KUKA KRL program: vw_sz_usr_s.src, vw_sz_usr_s.dat

--- vw_sz_usr_s.src ---
&ACCESS RV
&REL 203
&PARAM DISKPATH = VW_User/Applikation/S_Zange
&PARAM TPVW_VERSION = 8.3.0
DEF vw_sz_usr_s( )
;
;*-----------------------------------------------------*
;*Technologiepaket S_Zangen                            *
;*                                                     *
;*Konzernstandard                                      *
;*Bearbeiter: W. Lehmeier I/PG-C61                     *
;*                                                     *
;* Erstellt am:                                        *
;* 2015.02.19 LE                                       *
;* 2017.01.26 MBA Anpassung Teachfunktion KE           *
;* 2017.02.03 MBA Mit_BM1 bei BM2 korrigiert           *
;*            Zangenfkt. bei BM2 korrigiert            *
;* 2017.09.26 LZ "F_SZ_POT_Fra=838" bei POT gegen      *
;*            "Prog_Nr_SZ#>98" getauscht               *
;*                                                     *
;*------------------------------------------------------
;
END
;
;FOLD INIT S_Zangen
GLOBAL DEF SZ_INIT( )
INT i
;
;FOLD Version Techpaket
Tech_S_Zangen.Name[]="KS24.01.008_170926"
;ENDFOLD
;
;FOLD Vorbesetzung Meldungsausgabe
FOR i = 1 TO 100
  n_SZS_Handle[i]=-1
  n_SZR_Handle[i]=-1
ENDFOR
;ENDFOLD
;
;FOLD TimerInit
FOR i = 1 TO 3
  LBitTimeCnt[i] = $Rob_Timer
ENDFOR
;ENDFOLD
;
; Zaehle Flags fuer q-Tool
;SZ1
IF $Flag[F_QT_SZ1_VW] THEN
  Q_T_SZ1_VW=Q_T_SZ1_VW+1
ENDIF
IF $Flag[F_QT_SZ1_Fe] THEN
  Q_T_SZ1_Fe=Q_T_SZ1_Fe+1
ENDIF
IF $Flag[F_QT_SZ1_kD] THEN
  Q_T_SZ1_kD=Q_T_SZ1_kD+1
ELSE
  Q_T_SZ1_kD=0
ENDIF
;
;SZ2
IF $Flag[F_QT_SZ2_VW] THEN
  Q_T_SZ2_VW=Q_T_SZ2_VW+1
ENDIF
IF $Flag[F_QT_SZ2_Fe] THEN
  Q_T_SZ2_Fe=Q_T_SZ2_Fe+1
ENDIF
IF $Flag[F_QT_SZ2_kD] THEN
  Q_T_SZ2_kD=Q_T_SZ2_kD+1
ELSE
  Q_T_SZ2_kD=0
ENDIF
;SZ3
;
IF $Flag[F_QT_SZ3_VW] THEN
  Q_T_SZ3_VW=Q_T_SZ3_VW+1
ENDIF
IF $Flag[F_QT_SZ3_Fe] THEN
  Q_T_SZ3_Fe=Q_T_SZ3_Fe+1
ENDIF
IF $Flag[F_QT_SZ3_kD] THEN
  Q_T_SZ3_kD=Q_T_SZ3_kD+1
ELSE
  Q_T_SZ3_kD=0
ENDIF
;
; Zaehlergrenze damit kein ueberlauf entsteht
IF Q_T_SZ1_VW>1000000 THEN
  Q_T_SZ1_VW=0
ENDIF
IF Q_T_SZ1_Fe>1000000 THEN
  Q_T_SZ1_Fe=0
ENDIF
IF Q_T_SZ1_kD>1000000 THEN
  Q_T_SZ1_kD=0
ENDIF
IF Q_T_SZ2_VW>1000000 THEN
  Q_T_SZ2_VW=0
ENDIF
IF Q_T_SZ2_Fe>1000000 THEN
  Q_T_SZ2_Fe=0
ENDIF
IF Q_T_SZ2_kD>1000000 THEN
  Q_T_SZ2_kD=0
ENDIF
IF Q_T_SZ3_VW>1000000 THEN
  Q_T_SZ3_VW=0
ENDIF
IF Q_T_SZ3_Fe>1000000 THEN
  Q_T_SZ3_Fe=0
ENDIF
IF Q_T_SZ3_kD>1000000 THEN
  Q_T_SZ3_kD=0
ENDIF
;
$FLAG[F_QT_SZ1_VW]=FALSE
$FLAG[F_QT_SZ1_Fe]=FALSE
$FLAG[F_QT_SZ1_kD]=FALSE
$FLAG[F_QT_SZ2_VW]=FALSE
$FLAG[F_QT_SZ2_Fe]=FALSE
$FLAG[F_QT_SZ2_kD]=FALSE
$FLAG[F_QT_SZ3_VW]=FALSE
$FLAG[F_QT_SZ3_Fe]=FALSE
$FLAG[F_QT_SZ3_kD]=FALSE
;
;FOLD Vorbesetzung SZ1-3
IF $PRO_STATE1==#P_FREE THEN
  IF ($softplcint[2]>0) AND (NOT Docking OR DKSZ_stat_SZ) THEN
    I_SZ2_bereit=865
    O_SZ2_FRG=875
    I_SZ2_aktiv=875
    O_SZ2_SPos_g=876
    I_SZ2_IPos_g=876
    I_SZ2_F_Ziel=933
    ;Docking Downgrade
    bhf3_belegt=4081
    bhf4_belegt=4081
  ENDIF
  IF ($softplcint[3]>0) AND (NOT Docking OR DKSZ_stat_SZ) THEN
    I_SZ3_bereit=1025
    O_SZ3_FRG=1035
    I_SZ3_aktiv=1035
    O_SZ3_SPos_g=1036
    I_SZ3_IPos_g=1036
    I_SZ3_F_Ziel=1093
    ;Docking Downgrade
    bhf3_belegt=559
    bhf4_belegt=4081
  ENDIF
  IF Docking AND NOT DOCK_SP AND NOT DKSZ_stat_SZ THEN
    I_SZ2_bereit=4081
    O_SZ2_FRG=3658
    I_SZ2_aktiv=4082
    O_SZ2_SPos_g=3658
    I_SZ2_IPos_g=4081
    I_SZ2_F_Ziel=4082
    I_SZ3_bereit=4081
    O_SZ3_FRG=3658
    I_SZ3_aktiv=4082
    O_SZ3_SPos_g=3658
    I_SZ3_IPos_g=4081
    I_SZ3_F_Ziel=4082
    ;Docking Downgrade
    IF (AX_SIM_ON=='B000111000000') OR (AX_SIM_ON=='B001110000000') THEN
      bhf3_belegt=559
    ENDIF
    IF (AX_SIM_ON=='B001111000000') OR (AX_SIM_ON=='B011110000000') THEN
      bhf4_belegt=560
    ENDIF
  ENDIF
ENDIF
;ENDFOLD (Vorbesetzung SZ1-3)
;
;Ausgleichsfunktion initialisieren
R1AusgleichFunktion=0
GunBal_Halt=FALSE
;
;Hilfsflag fuer SZ-AH-Kompensation ausschalten
$FLAG[F_SZ_AH_KOMP]=FALSE
;Hilfsflag fuer SZ_Schliessen ausschalten
$FLAG[F_SZ1_Schliess]=FALSE
$FLAG[F_SZ2_Schliess]=FALSE
$FLAG[F_SZ3_Schliess]=FALSE
;
;Initiallisierung Kappenstandzeit Z1-3
FOR i = 1 TO 10
  IF (ReserveReal[i]==0.0) THEN
    ReserveReal[i]=28.0
  ENDIF
ENDFOR
;
END
;ENDFOLD
;
;-----------------------------------------------------------
;FOLD SAW S_Zangen
GLOBAL DEF SZ_SAW( )
INT i
;
;FOLD S_Zangen 1-3
IF ($softplcint[1]>0) AND NOT ($OUT[O_SZ1_Re_aus] OR $OUT[O_SZ1_MnFrae] OR $OUT[O_Kb1_MnFrae] OR $FLAG[F_SZ1_FRG_FR]) THEN
  $OUT[O_SZ1_S_TPos]=FALSE
  $OUT[O_SZ1_ref]=FALSE
  $OUT[O_SZ1_FRG]=FALSE
  $OUT[O_SZ1_auf]=FALSE
  $OUT[O_SZ1_zu]=FALSE
  $OUT[O_SZ1_t_auf]=FALSE
  $OUT[O_SZ1_t_zu]=FALSE
  IF Mit_Komb_ST1 THEN
    $OUT[O_Kb1_t_auf]=FALSE
    $OUT[O_Kb1_t_zu]=FALSE
  ENDIF
ENDIF
IF ($softplcint[2]>0) AND NOT ($OUT[O_SZ2_Re_aus] OR $OUT[O_SZ2_MnFrae] OR $OUT[O_Kb2_MnFrae] OR $FLAG[F_SZ2_FRG_FR]) THEN
  $OUT[O_SZ2_S_TPos]=FALSE
  $OUT[O_SZ2_ref]=FALSE
  $OUT[O_SZ2_FRG]=FALSE
  $OUT[O_SZ2_auf]=FALSE
  $OUT[O_SZ2_zu]=FALSE
  $OUT[O_SZ2_t_auf]=FALSE
  $OUT[O_SZ2_t_zu]=FALSE
  IF Mit_Komb_ST2 THEN
    $OUT[O_Kb2_t_auf]=FALSE
    $OUT[O_Kb2_t_zu]=FALSE
  ENDIF
ENDIF
IF ($softplcint[3]>0) AND NOT ($OUT[O_SZ3_Re_aus] OR $OUT[O_SZ3_MnFrae] OR $OUT[O_Kb3_MnFrae] OR $FLAG[F_SZ3_FRG_FR]) THEN
  $OUT[O_SZ3_S_TPos]=FALSE
  $OUT[O_SZ3_ref]=FALSE
  $OUT[O_SZ3_FRG]=FALSE
  $OUT[O_SZ3_auf]=FALSE
  $OUT[O_SZ3_zu]=FALSE
  $OUT[O_SZ3_t_auf]=FALSE
  $OUT[O_SZ3_t_zu]=FALSE
  IF Mit_Komb_ST3 THEN
    $OUT[O_Kb3_t_auf]=FALSE
    $OUT[O_Kb3_t_zu]=FALSE
  ENDIF
ENDIF
HAND_FKT1=FALSE
HAND_FKT2=FALSE
;
;SZ Ausgleich durch Roboter
IF R1AusgleichFunktion>0 THEN
  R1AusgleichFunktion=0
  S_Zangen_Msg(20,#NotifyMsg)
ENDIF
GunBal_Halt=FALSE
;
;Hilfsflag fuer SZ-AH-Kompensation ausschalten
$FLAG[F_SZ_AH_KOMP]=FALSE
;Hilfsflag fuer SZ_Schliessen ausschalten
$FLAG[F_SZ1_Schliess]=FALSE
$FLAG[F_SZ2_Schliess]=FALSE
$FLAG[F_SZ3_Schliess]=FALSE
;ENDFOLD
;
END
;ENDFOLD
;
;-----------------------------------------------------------
;FOLD RESET S_Zangen
GLOBAL DEF SZ_RESET( )
INT i
;
;FOLD S_Zangen 1-3
IF (($mode_op==#T1) OR ($mode_op==#T2)) THEN
  $softplcint[20]=0
  IF ($softplcint[1]>0) THEN
    $FLAG[F_SZ_AH_KOMP]=FALSE
    $OUT[O_SZ1_FRG]=FALSE
    $OUT[O_SZ1_S_TPos]=FALSE
    $OUT[O_SZ1_ref]=FALSE
    $OUT[O_SZ1_auf]=FALSE
    $OUT[O_SZ1_zu]=FALSE
    $OUT[O_SZ1_t_auf]=FALSE
    $OUT[O_SZ1_t_zu]=FALSE
    $OUT[O_SZ1_MvFrae]=FALSE
    $OUT[O_SZ1_MnFrae]=FALSE
    IF Mit_Komb_ST1 THEN
      $OUT[O_Kb1_t_auf]=FALSE
      $OUT[O_Kb1_t_zu]=FALSE
    ENDIF
  ENDIF
;
  IF ($softplcint[2]>0) THEN
    $OUT[O_SZ2_FRG]=FALSE
    $OUT[O_SZ2_S_TPos]=FALSE
    $OUT[O_SZ2_ref]=FALSE
    $OUT[O_SZ2_auf]=FALSE
    $OUT[O_SZ2_zu]=FALSE
    $OUT[O_SZ2_t_auf]=FALSE
    $OUT[O_SZ2_t_zu]=FALSE
    $OUT[O_SZ2_MvFrae]=FALSE
    $OUT[O_SZ2_MnFrae]=FALSE
    IF Mit_Komb_ST2 THEN
      $OUT[O_Kb2_t_auf]=FALSE
      $OUT[O_Kb2_t_zu]=FALSE
    ENDIF
  ENDIF
;
  IF ($softplcint[3]>0) THEN
    $OUT[O_SZ3_FRG]=FALSE
    $OUT[O_SZ3_S_TPos]=FALSE
    $OUT[O_SZ3_ref]=FALSE
    $OUT[O_SZ3_auf]=FALSE
    $OUT[O_SZ3_zu]=FALSE
    $OUT[O_SZ3_t_auf]=FALSE
    $OUT[O_SZ3_t_zu]=FALSE
    $OUT[O_SZ3_MvFrae]=FALSE
    $OUT[O_SZ3_MnFrae]=FALSE
    IF Mit_Komb_ST3 THEN
      $OUT[O_Kb3_t_auf]=FALSE
      $OUT[O_Kb3_t_zu]=FALSE
    ENDIF
  ENDIF
;
  ;SZ Ausgleich durch Roboter
  R1AusgleichFunktion=0
  GunBal_Halt=FALSE
;
  ;Hilfsflag fuer SZ-AH-Kompensation ausschalten
  $FLAG[F_SZ_AH_KOMP]=FALSE
  ;Hilfsflag fuer SZ_Schliessen ausschalten
  $FLAG[F_SZ1_Schliess]=FALSE
  $FLAG[F_SZ2_Schliess]=FALSE
  $FLAG[F_SZ3_Schliess]=FALSE
ENDIF ;(SZ_VORHANDEN)
;ENDFOLD
;
END
;ENDFOLD
;
;-----------------------------------------------------------
;FOLD CANCEL S_Zangen
GLOBAL DEF SZ_CANCEL( )
INT i
;
;FOLD S_Zangen 1-3
IF (($mode_op==#T1) OR ($mode_op==#T2)) THEN
  $softplcint[20]=0
  IF ($softplcint[1]>0) THEN
    $FLAG[F_SZ_AH_KOMP]=FALSE
    $OUT[O_SZ1_FRG]=FALSE
    $OUT[O_SZ1_S_TPos]=FALSE
    $OUT[O_SZ1_ref]=FALSE
    $OUT[O_SZ1_auf]=FALSE
    $OUT[O_SZ1_zu]=FALSE
    $OUT[O_SZ1_t_auf]=FALSE
    $OUT[O_SZ1_t_zu]=FALSE
    $OUT[O_SZ1_MvFrae]=FALSE
    $OUT[O_SZ1_MnFrae]=FALSE
    IF Mit_Komb_ST1 THEN
      $OUT[O_Kb1_t_auf]=FALSE
      $OUT[O_Kb1_t_zu]=FALSE
    ENDIF
  ENDIF
;
  IF ($softplcint[2]>0) THEN
    $OUT[O_SZ2_FRG]=FALSE
    $OUT[O_SZ2_S_TPos]=FALSE
    $OUT[O_SZ2_ref]=FALSE
    $OUT[O_SZ2_auf]=FALSE
    $OUT[O_SZ2_zu]=FALSE
    $OUT[O_SZ2_t_auf]=FALSE
    $OUT[O_SZ2_t_zu]=FALSE
    $OUT[O_SZ2_MvFrae]=FALSE
    $OUT[O_SZ2_MnFrae]=FALSE
    IF Mit_Komb_ST2 THEN
      $OUT[O_Kb2_t_auf]=FALSE
      $OUT[O_Kb2_t_zu]=FALSE
    ENDIF
  ENDIF
;
  IF ($softplcint[3]>0) THEN
    $OUT[O_SZ3_FRG]=FALSE
    $OUT[O_SZ3_S_TPos]=FALSE
    $OUT[O_SZ3_ref]=FALSE
    $OUT[O_SZ3_auf]=FALSE
    $OUT[O_SZ3_zu]=FALSE
    $OUT[O_SZ3_t_auf]=FALSE
    $OUT[O_SZ3_t_zu]=FALSE
    $OUT[O_SZ3_MvFrae]=FALSE
    $OUT[O_SZ3_MnFrae]=FALSE
    IF Mit_Komb_ST3 THEN
      $OUT[O_Kb3_t_auf]=FALSE
      $OUT[O_Kb3_t_zu]=FALSE
    ENDIF
  ENDIF
;
  ;SZ Ausgleich durch Roboter
  R1AusgleichFunktion=0
  GunBal_Halt=FALSE
;
  ;Hilfsflag fuer SZ-AH-Kompensation ausschalten
  $FLAG[F_SZ_AH_KOMP]=FALSE
  ;Hilfsflag fuer SZ_Schliessen ausschalten
  $FLAG[F_SZ1_Schliess]=FALSE
  $FLAG[F_SZ2_Schliess]=FALSE
  $FLAG[F_SZ3_Schliess]=FALSE
ENDIF ;(SZ_VORHANDEN)
;ENDFOLD
;
END
;ENDFOLD
;
;-----------------------------------------------------------
;FOLD LOOP S_Zange 1
GLOBAL DEF SZ1_LOOP( )
;
;SZ 1 Funktionstest ohne Bauteil
IF Mit_Komb_ST1 THEN
  $OUT[O_Kb1_FToBT]=$IN[I_FT_o_BT]
  IF (Prog_Nr_Kb1<99) AND ($FLAG[F_SZ1_FRG_FR] OR $OUT[O_R_Wart] OR $OUT[O_R_WartB]) THEN
    Fzg_Typ_SZ1=0
  ENDIF
ELSE
  $OUT[O_SZ1_FToBT]=$IN[I_FT_o_BT] AND (Prog_Nr_SZ1>98)
  IF (Prog_Nr_SZ1<99) AND ($FLAG[F_SZ1_FRG_FR] OR $OUT[O_R_Wart] OR $OUT[O_R_WartB]) THEN
    Fzg_Typ_SZ1=0
	 SK1_Fzg_Typ=0
  ENDIF
ENDIF
;
;SZ 1 Anwahl Energiesparmodus
$OUT[O_SZ1_E_Mode] = (($Brake_Sig==0) AND $timer_flag[TimerNr_E_Mo] AND e_Mode_Hilf2)
;
;FOLD SZ Betriebsarten
;BA-Hand an SZ 1 setzen
IF $OUT[O_R_Hand] AND (NOT $COULD_START_MOTION OR HAND_FKT2) THEN
  $OUT[O_SZ1_R_Hand]=TRUE
  $OUT[O_SZ1_R_Auto]=FALSE
ENDIF
;
;BA-AUTO an SZ 1 setzen
IF $OUT[O_R_Hand] AND NOT HAND_FKT2 AND ($OUT[O_R_Proz_akt] OR $OUT[O_R_bewegt] OR TAST_AKTIV_1 OR TAST_AKTIV_2 OR TAST_AKTIV_3 OR HAND_FKT1) AND (R1AusgleichFunktion==0) OR $OUT[O_R_Auto] THEN
  $OUT[O_SZ1_R_Hand]=FALSE
  $OUT[O_SZ1_R_Auto]=TRUE
ENDIF
;ENDFOLD
;
;SZ 1 mit EK-Verschleisswert
$OUT[O_SZ1_Mit_EK]=TRUE
;
;SZ 1 ohne Kraft
IF $IN[I_SZ1_oh_Kra] THEN
  $OUT[O_SZ1_oh_Kra]=TRUE
ELSE
  $OUT[O_SZ1_oh_Kra]=FALSE
ENDIF
;
;SZ Kraftvorgabe in Hand
IF NOT Mit_Komb_ST1  THEN
  IF $OUT[O_R_Hand] AND $FLAG[F_o_Prozess] THEN
    SZ1_Kraft_Soll = M_Kraft_Soll
  ELSE
    SZ1_Kraft_Soll = SK1_Kraft_Soll
  ENDIF
ENDIF
;ENDFOLD
;
;Kompensation der EK durch Roboter
IF AH_Komp AND NOT $FLAG[F_SZ1_m_Komp] AND NOT Mit_Komb_ST1 THEN
  $OUT[O_SZ1_m_RKom]=TRUE
ELSE
  $OUT[O_SZ1_m_RKom]=FALSE
ENDIF
;
;Quittierung Stoerung
IF Mit_Komb_ST1 THEN
  $OUT[O_Kb1_Fe_Res]=($IN[I_Kb1_Sammel] AND $IN[I_R_Quit_St]) OR (($IN[I_R_Quit_Wei] OR $FLAG[F_SZ_Fe_Res]) AND $IN[I_Kb1_Sammel])
ELSE
  $OUT[O_SZ1_Fe_Res]=($IN[I_SZ1_Sammel] AND $IN[I_R_Quit_St]) OR (($IN[I_R_Quit_Wei] OR $FLAG[F_SZ_Fe_Res]) AND $IN[I_SZ1_Sammel])
ENDIF
;
;Ausgabe Statusmeldungen an BMS
IF Mit_Komb_ST1 THEN
  ;Vorwahl mit Strom
  $OUT[O_Kb1_m_Stro]=NOT $IN[I_Kb1_o_Schw] AND NOT $FLAG[F_o_Prozess]
  ;Start Protokoll
  $OUT[O_Kb1_Protok]=$IN[I_Kb1_Protok]
  ;Vorwarnung Zange
  $OUT[O_Kb1_W_SZ]=($IN[I_SZ1_W_SZ] OR (Q_T_SZ1_VW>3) OR (Q_T_SZ1_kD>50))
  ;Warnung Schmierung
  $OUT[O_Kb1_W_Schm]=$IN[I_SZ1_W_Schm]
  ;Fraesanfrage
  $OUT[O_Kb1_FrAnf]=$OUT[O_R_Auto] AND $IN[I_Kb1_FrAnf]
  ;Vorwarnung Kappenstandzeit
  $OUT[O_Kb1_V_Stdm]=($IN[I_Kb1_V_Stdm] OR B_SK1_V_Stdm)
  ;Maximale Kappenstandzeit
  $OUT[O_Kb1_M_Stdm]=($IN[I_SZ1_F_Geom] OR $IN[I_Kb1_M_Stdm] OR B_SK1_M_Stdm OR $FLAG[F_SK1_max_SZ1] OR $FLAG[F_SK1_max_SZ2] OR $FLAG[F_SK1_max_SZ3] OR $FLAG[F_SK1_max_SZ4])
  ;Kraftaufbau zu lange
  $OUT[O_Kb1_F_Kraf]=$OUT[O_R_Auto] AND $IN[I_SZ1_F_Kraf]
  ;Punktanwahlfehler
  $OUT[O_Kb1_F_Prog]=$OUT[O_R_Auto] AND $IN[I_SZ1_F_Prog]
  ;Zielposition ungueltig
  $OUT[O_Kb1_F_Ziel]=$OUT[O_R_Auto] AND $IN[I_SZ1_F_Ziel]
  ;Bauteilfehler
  $OUT[O_Kb1_F_Baut]=$OUT[O_R_Auto] AND $IN[I_SZ1_F_Baut]
  ;Zange geht schwer
  $OUT[O_Kb1_F_schw]=$OUT[O_R_Auto] AND $IN[I_SZ1_F_schw]
  ;Fraesen n.i.O.
  $OUT[O_Kb1_F_Frae]=$OUT[O_R_Auto] AND $IN[I_SZ1_F_Frae]
  ;Fehler Kappenverschleiss
  $OUT[O_Kb1_F_KaVe]=$OUT[O_R_Auto] AND ($IN[I_SZ1_F_Kapp] OR $FLAG[F_SZ1_Kapp1] OR $FLAG[F_SZ1_Kapp2] OR $FLAG[F_SZ1_Kapp3] OR $FLAG[F_SZ1_Kapp4])
  ;Fehler Geometrie
  $OUT[O_Kb1_F_Geom]=$OUT[O_R_Auto] AND $IN[I_SZ1_F_Geom]
  ;Schleppfehler
  $OUT[O_Kb1_Schlep]=$OUT[O_R_Auto] AND $IN[I_SZ1_F_Schl]
  ;Fehler Ausgleichssystem
  $OUT[O_Kb1_F_Ausg]=$OUT[O_R_Auto] AND ($IN[I_SZ1_F_Ausg] OR (Q_T_SZ1_Fe>3))
  ;Fehler Steuerung/Regler
  $OUT[O_Kb1_F_Steu]=$OUT[O_R_Auto] AND $COULD_START_MOTION AND $IN[I_SZ1_F_Steu]
  ;Fehler Temperatur Trafo
  $OUT[O_Kb1_FT_Tra]=$OUT[O_R_Auto] AND $IN[I_SZ1_F_Traf]
  ;Fehler Temperatur Motor
  $OUT[O_Kb1_FT_Mot]=$OUT[O_R_Auto] AND $IN[I_SZ1_F_Mot]
  ;Schweissung i.O
  $OUT[O_Kb1_WPS_io]=$OUT[O_R_Auto] AND NOT $FLAG[F_SK1_S_niO]
  ;Schweissung n.i.O
  $OUT[O_Kb1_WP_nio]=$OUT[O_R_Auto] AND $FLAG[F_SK1_S_niO]
  ;Warngrenze verletzt in Folge
  $OUT[O_Kb1_W_Folg]=$OUT[O_R_Auto] AND $IN[I_Kb1_W_Folg]
  ;Phasenueberwachung
  $OUT[O_Kb1_Ph_nio]=$OUT[O_R_Auto] AND $IN[I_Kb1_Ph_nio]
  ;Ueberstrom Primaerseite
  $OUT[O_Kb1_Primae]=$OUT[O_R_Auto] AND $IN[I_Kb1_Primae]
  ;Fehler Stromsensor
  $OUT[O_Kb1_F_Stro]=$OUT[O_R_Auto] AND $IN[I_Kb1_F_Stro]
  ;Fehler Spannungssensor
  $OUT[O_Kb1_F_Span]=$OUT[O_R_Auto] AND $IN[I_Kb1_F_Span]
  ;Überstrom 24 V DC
  $OUT[O_Kb1_24V]=$OUT[O_R_Auto] AND $IN[I_Kb1_24V]
  ;Uebertemperatur Inverter
  $OUT[O_Kb1_Invert]=$OUT[O_R_Auto] AND $IN[I_Kb1_Invert]
  ;Sammelstoerung
  $OUT[O_Kb1_Sammel]=$OUT[O_R_Auto] AND $COULD_START_MOTION AND ($IN[I_Kb1_Sammel] OR $FLAG[F_SZ1_Sammel] OR $FLAG[F_SK1_Sammel] OR SZ_LBitFeh[1]) AND $timer_flag[TimerNr_Ein]
ELSE
  ;Vorwarnung Zange
  $OUT[O_SZ1_W_SZ]=($IN[I_SZ1_W_SZ] OR (Q_T_SZ1_VW>3) OR (Q_T_SZ1_kD>50))
  ;Warnung Schmierung
  $OUT[O_SZ1_W_Schm]=$IN[I_SZ1_W_Schm]
  ;Kraftaufbau zu lange
  $OUT[O_SZ1_F_Kraf]=$OUT[O_R_Auto] AND $IN[I_SZ1_F_Kraf]
  ;Programmfehler/falsche Kraftvorgabe
  $OUT[O_SZ1_F_Prog]=$OUT[O_R_Auto] AND $IN[I_SZ1_F_Prog]
  ;Zielposition ungueltig
  $OUT[O_SZ1_F_Ziel]=$OUT[O_R_Auto] AND $IN[I_SZ1_F_Ziel]
  ;Bauteilfehler
  $OUT[O_SZ1_F_Baut]=$OUT[O_R_Auto] AND $IN[I_SZ1_F_Baut]
  ;Zange geht schwer
  $OUT[O_SZ1_F_schw]=$OUT[O_R_Auto] AND $IN[I_SZ1_F_schw]
  ;Fraesen n.i.O.
  $OUT[O_SZ1_F_Frae]=$OUT[O_R_Auto] AND $IN[I_SZ1_F_Frae]
  ;Fehler Kappenverschleiss/Geometrie
  $OUT[O_SZ1_F_Geom]=$OUT[O_R_Auto] AND ($IN[I_SZ1_F_Kapp] OR $IN[I_SZ1_F_Geom] OR $FLAG[F_SZ1_Kapp1] OR $FLAG[F_SZ1_Kapp2] OR $FLAG[F_SZ1_Kapp3] OR $FLAG[F_SZ1_Kapp4])
  ;Fehler Ausgleichssystem
  $OUT[O_SZ1_F_Ausg]=$OUT[O_R_Auto] AND ($IN[I_SZ1_F_Ausg] OR (Q_T_SZ1_Fe>3))
  ;Fehler Steuerung/Regler
  $OUT[O_SZ1_F_Steu]=$OUT[O_R_Auto] AND $COULD_START_MOTION AND $IN[I_SZ1_F_Steu]
  ;Fehler Temperatur Motor/Trafo
  $OUT[O_SZ1_F_Temp]=$OUT[O_R_Auto] AND ($IN[I_SZ1_F_Traf] OR $IN[I_SZ1_F_Mot])
  ;Sammelstoerung
  $OUT[O_SZ1_Sammel]=$OUT[O_R_Auto] AND $COULD_START_MOTION AND ($IN[I_SZ1_Sammel] OR $FLAG[F_SZ1_Sammel] OR SZ_LBitFeh[1]) AND $timer_flag[TimerNr_Ein]
ENDIF
;
;Ausgabe Zangencode
IF NOT Docking OR (Docking AND NOT Dock_SZ) THEN
  IF Mit_Komb_ST THEN
    Kb1_ZCode=1
  ELSE
    EZ1_ZCode=1
  ENDIF
ENDIF
;
;FOLD SZ-Tastbetrieb ruecksetzen
IF Mit_Komb_ST1 THEN
  Temp_Komb_1=($OUT[O_Kb1_t_zu] OR $OUT[O_Kb1_t_auf])
ENDIF
IF $OUT[O_R_Hand] AND TAST_AKTIV_1 AND NOT $OUT[O_SZ1_t_auf] AND NOT $OUT[O_SZ1_t_zu] AND NOT Temp_Komb_1 THEN
  TAST_AKTIV_1=FALSE
  $OUT[O_SZ1_FRG]=FALSE
  schleppfehler=TRUE
  sf_prog_status=#user_act
  $OUT[O_SZ1_SPos_g]=FALSE
ENDIF
;ENDFOLD
;
;FOLD SZ INIT Zangenfunktion
IF $OUT[O_R_Hand] AND NOT $OUT[O_R_Auto] AND $COULD_START_MOTION AND ((NOT $OUT[O_R_Proz_akt] AND NOT $OUT[O_R_bewegt]) OR (R1AusgleichFunktion>0)) THEN
  IF Mit_Komb_ST1 THEN
    Temp_Komb_1=$OUT[O_Kb1_t_zu]
  ENDIF
  IF ($OUT[O_SZ1_S_TPos] OR $OUT[O_SZ1_ref] OR $OUT[O_SZ1_auf] OR $OUT[O_SZ1_zu] OR Temp_Komb_1 OR $OUT[O_SZ1_t_auf] OR $OUT[O_SZ1_t_zu] OR $OUT[O_SZ1_Teach] OR $OUT[O_SZ1_D_Auf] OR $OUT[O_SZ1_Du_Zu]) THEN
    CheckZangenFunktion()
    Zangenfunktion()
  ENDIF
ELSE
  IF $OUT[O_SZ1_Teach] OR $OUT[O_SZ1_D_Auf] OR $OUT[O_SZ1_Du_Zu] THEN
    $OUT[O_SZ1_Teach]=FALSE
    $OUT[O_SZ1_D_Auf]=FALSE
    $OUT[O_SZ1_Du_Zu]=FALSE
    S_Zangen_Msg(34,#NotifyMsg)
  ENDIF
ENDIF
;ENDFOLD
;
;FOLD Ruecksetzen Zangenfunktion
IF ($OUT[O_R_Hand] AND ($PRO_MODE1==#BSTEP)) OR ($OUT[O_R_Hand] AND NOT $FLAG[F_SZ_AH_KOMP] AND $OUT[O_R_bewegt] AND (R1AusgleichFunktion==0)) OR ($OUT[O_R_Hand] AND NOT $COULD_START_MOTION AND (HAND_FKT1 OR HAND_FKT2)) THEN
  IF NOT ($OUT[O_SZ1_Re_aus] OR $OUT[O_SZ1_MnFrae] OR $OUT[O_Kb1_MnFrae] OR $FLAG[F_SZ1_FRG_FR]) THEN
    $OUT[O_SZ1_S_TPos]=FALSE
    $OUT[O_SZ1_ref]=FALSE
    $OUT[O_SZ1_FRG]=FALSE
    $OUT[O_SZ1_auf]=FALSE
    $OUT[O_SZ1_zu]=FALSE
    $OUT[O_SZ1_t_auf]=FALSE
    $OUT[O_SZ1_t_zu]=FALSE
    IF Mit_Komb_ST1 THEN
      $OUT[O_Kb1_t_auf]=FALSE
      $OUT[O_Kb1_t_zu]=FALSE
    ENDIF
  ENDIF
  HAND_FKT1=FALSE
  HAND_FKT2=FALSE
ENDIF
;ENDFOLD
;
;FOLD EZ Oeffnungsmass beim Schwenken pruefen
;EZ/SP1
IF ($softplcint[1]>0) AND $OUT[O_SZ1_FRG] AND (Varstate("act_P1")==#initialized) THEN
  IF ($softplcint[1]==7) THEN
    $FLAG[F_SZ1_Oeff_iO]=(act_P1.E1>=$COUNT_I[60])
  ENDIF
  IF ($softplcint[1]==8) THEN
    $FLAG[F_SZ1_Oeff_iO]=(act_P1.E2>=$COUNT_I[60])
  ENDIF
ELSE
  $FLAG[F_SZ1_Oeff_iO]=FALSE
ENDIF
;ENDFOLD
;
;FOLD EZ Position nach Messen und Fraesen pruefen
$FLAG[Mit_Anf_Pos]=TRUE
;EZ/SP1
IF ($softplcint[1]>0) AND $FLAG[F_SZ_Anf_Pos] AND $OUT[O_SZ1_FRG] AND (Varstate("act_P1")==#initialized) THEN
  $FLAG[F_SZ_Anf_Pos]=FALSE
  IF ($softplcint[1]==7) THEN
    $FLAG[F_SZ1_Pos_iO]=((sig1_istpos>=((act_P1.E1*10)-140)) AND (sig1_istpos<=((act_P1.E1*10)+140)))
  ENDIF
  IF ($softplcint[1]==8) THEN
    $FLAG[F_SZ1_Pos_iO]=((sig1_istpos>=((act_P1.E2*10)-140)) AND (sig1_istpos<=((act_P1.E2*10)+140)))
  ENDIF
  IF ($softplcint[1]==9) THEN
    $FLAG[F_SZ1_Pos_iO]=((sig1_istpos>=((act_P1.E3*10)-140)) AND (sig1_istpos<=((act_P1.E3*10)+140)))
  ENDIF
  IF ($softplcint[1]==10) THEN
    $FLAG[F_SZ1_Pos_iO]=((sig1_istpos>=((act_P1.E4*10)-140)) AND (sig1_istpos<=((act_P1.E4*10)+140)))
  ENDIF
  IF ($softplcint[1]==11) THEN
    $FLAG[F_SZ1_Pos_iO]=((sig1_istpos>=((act_P1.E5*10)-140)) AND (sig1_istpos<=((act_P1.E5*10)+140)))
  ENDIF
ENDIF
;ENDFOLD
;
;FOLD Ruecksetzen Ausgabe max. Kappenverschleiss
IF $OUT[O_SZ1_KW_io] THEN
  B_SK1_M_Stdm = FALSE
  B_SK1_V_Stdm = FALSE
  B_SK1_FRG_Ge = TRUE
  IF (($softplcint[1]==7) OR ($softplcint[1]==8)) AND (Dock_Z1==TRUE) THEN
    B_SK1_FRG_G1 = TRUE
  ENDIF
  IF (($softplcint[1]==8) OR ($softplcint[1]==9)) AND (Dock_Z2==TRUE) THEN
    B_SK1_FRG_G2 = TRUE
  ENDIF
  IF (($softplcint[1]==9) OR ($softplcint[1]==10)) AND (Dock_Z3==TRUE) THEN
    B_SK1_FRG_G3 = TRUE
  ENDIF
  IF (($softplcint[1]==10) OR ($softplcint[1]==11)) AND (Dock_Z4==TRUE) THEN
    B_SK1_FRG_G4 = TRUE
  ENDIF
ENDIF
;ENDFOLD
;
;FOLD Lebensbit
IF Mit_Komb_ST1 THEN
  L_Bit_Kombi(1)
ELSE
  L_Bit_SZ(1)
ENDIF
;ENDFOLD
;
END
;ENDFOLD
;
;-----------------------------------------------------------
;FOLD LOOP S_Zange 2
GLOBAL DEF SZ2_LOOP( )
;
;SZ 2 Funktionstest ohne Bauteil
IF Mit_Komb_ST2 THEN
  $OUT[O_Kb2_FToBT]=$IN[I_FT_o_BT]
  IF (Prog_Nr_Kb2<99) AND ($FLAG[F_SZ2_FRG_FR] OR $OUT[O_R_Wart] OR $OUT[O_R_WartB]) THEN
    Fzg_Typ_SZ2=0
  ENDIF
ELSE
  $OUT[O_SZ2_FToBT]=$IN[I_FT_o_BT] AND (Prog_Nr_SZ2>98)
  IF (Prog_Nr_SZ2<99) AND ($FLAG[F_SZ2_FRG_FR] OR $OUT[O_R_Wart] OR $OUT[O_R_WartB]) THEN
    Fzg_Typ_SZ2=0
    SK2_Fzg_Typ=0
  ENDIF
ENDIF
;
;SZ 2 Anwahl Energiesparmodus
$OUT[O_SZ2_E_Mode] = (($Brake_Sig==0) AND $timer_flag[TimerNr_E_Mo] AND e_Mode_Hilf2)
;
;FOLD SZ Betriebsarten
;BA-Hand an SZ 2 setzen
IF $OUT[O_R_Hand] AND (NOT $COULD_START_MOTION OR HAND_FKT2) THEN
  $OUT[O_SZ2_R_Hand]=TRUE
  $OUT[O_SZ2_R_Auto]=FALSE
ENDIF
;
;BA-AUTO an SZ 2 setzen
IF $OUT[O_R_Hand] AND NOT HAND_FKT2 AND ($OUT[O_R_Proz_akt] OR $OUT[O_R_bewegt] OR TAST_AKTIV_1 OR TAST_AKTIV_2 OR TAST_AKTIV_3 OR HAND_FKT1) AND (R1AusgleichFunktion==0) OR $OUT[O_R_Auto] THEN
  $OUT[O_SZ2_R_Hand]=FALSE
  $OUT[O_SZ2_R_Auto]=TRUE
ENDIF
;ENDFOLD
;
;SZ 2 mit EK-Verschleisswert
$OUT[O_SZ2_Mit_EK]=TRUE
;
;SZ 2 ohne Kraft
IF $IN[I_SZ2_oh_Kra] THEN
  $OUT[O_SZ2_oh_Kra]=TRUE
ELSE
  $OUT[O_SZ2_oh_Kra]=FALSE
ENDIF
;
;SZ Kraftvorgabe in Hand
IF NOT Mit_Komb_ST2  THEN
  IF $OUT[O_R_Hand] AND $FLAG[F_o_Prozess] THEN
    SZ2_Kraft_Soll = M_Kraft_Soll
  ELSE
    IF Mit_2SZ_an_SK1 THEN
      SZ2_Kraft_Soll = SK1_Kraft_Soll
      $FLAG[F_2SZ_an_SK1]=TRUE
    ELSE
      SZ2_Kraft_Soll = SK2_Kraft_Soll
      $FLAG[F_2SZ_an_SK1]=FALSE
    ENDIF
  ENDIF
ENDIF
;
;Kompensation der EK durch Roboter
IF AH_Komp AND NOT $FLAG[F_SZ2_m_Komp] AND NOT Mit_Komb_ST2 THEN
  $OUT[O_SZ2_m_RKom]=TRUE
ELSE
  $OUT[O_SZ2_m_RKom]=FALSE
ENDIF
;
;Quittierung Stoerung
IF Mit_Komb_ST2 THEN
  $OUT[O_Kb2_Fe_Res]=($IN[I_Kb2_Sammel] AND $IN[I_R_Quit_St]) OR (($IN[I_R_Quit_Wei] OR $FLAG[F_SZ_Fe_Res]) AND $IN[I_Kb2_Sammel])
ELSE
  $OUT[O_SZ2_Fe_Res]=($IN[I_SZ2_Sammel] AND $IN[I_R_Quit_St]) OR (($IN[I_R_Quit_Wei] OR $FLAG[F_SZ_Fe_Res]) AND $IN[I_SZ2_Sammel])
ENDIF
;
;Ausgabe Statusmeldungen an BMS
IF Mit_Komb_ST2 THEN
  ;Vorwahl mit Strom
  $OUT[O_Kb2_m_Stro]=NOT $IN[I_Kb2_o_Schw] AND NOT $FLAG[F_o_Prozess]
  ;Start Protokoll
  $OUT[O_Kb2_Protok]=$IN[I_Kb2_Protok]
  ;Vorwarnung Zange
  $OUT[O_Kb2_W_SZ]=($IN[I_SZ2_W_SZ] OR (Q_T_SZ2_VW>3) OR (Q_T_SZ2_kD>50))
  ;Warnung Schmierung
  $OUT[O_Kb2_W_Schm]=$IN[I_SZ2_W_Schm]
  ;Fraesanfrage
  $OUT[O_Kb2_FrAnf]=$OUT[O_R_Auto] AND $IN[I_Kb2_FrAnf]
  ;Vorwarnung Kappenstandzeit
  $OUT[O_Kb2_V_Stdm]=($IN[I_Kb2_V_Stdm] OR B_SK2_V_Stdm)
  ;Maximale Kappenstandzeit
  $OUT[O_Kb2_M_Stdm]=($IN[I_SZ2_F_Geom] OR $IN[I_Kb2_M_Stdm] OR B_SK2_M_Stdm)
  ;Kraftaufbau zu lange
  $OUT[O_Kb2_F_Kraf]=$OUT[O_R_Auto] AND $IN[I_SZ2_F_Kraf]
  ;Punktanwahlfehler
  $OUT[O_Kb2_F_Prog]=$OUT[O_R_Auto] AND $IN[I_SZ2_F_Prog]
  ;Zielposition ungueltig
  $OUT[O_Kb2_F_Ziel]=$OUT[O_R_Auto] AND $IN[I_SZ2_F_Ziel]
  ;Bauteilfehler
  $OUT[O_Kb2_F_Baut]=$OUT[O_R_Auto] AND $IN[I_SZ2_F_Baut]
  ;Zange geht schwer
  $OUT[O_Kb2_F_schw]=$OUT[O_R_Auto] AND $IN[I_SZ2_F_schw]
  ;Fraesen n.i.O.
  $OUT[O_Kb2_F_Frae]=$OUT[O_R_Auto] AND $IN[I_SZ2_F_Frae]
  ;Fehler Kappenverschleiss
  $OUT[O_Kb2_F_KaVe]=$OUT[O_R_Auto] AND $IN[I_SZ2_F_Kapp]
  ;Fehler Geometrie
  $OUT[O_Kb2_F_Geom]=$OUT[O_R_Auto] AND $IN[I_SZ2_F_Geom]
  ;Schleppfehler
  $OUT[O_Kb2_Schlep]=$OUT[O_R_Auto] AND $IN[I_SZ2_F_Schl]
  ;Fehler Ausgleichssystem
  $OUT[O_Kb2_F_Ausg]=$OUT[O_R_Auto] AND ($IN[I_SZ2_F_Ausg] OR (Q_T_SZ2_VW>3))
  ;Fehler Steuerung/Regler
  $OUT[O_Kb2_F_Steu]=$OUT[O_R_Auto] AND $COULD_START_MOTION AND $IN[I_SZ2_F_Steu]
  ;Fehler Temperatur Trafo
  $OUT[O_Kb2_FT_Tra]=$OUT[O_R_Auto] AND $IN[I_SZ2_F_Traf]
  ;Fehler Temperatur Motor
  $OUT[O_Kb2_FT_Mot]=$OUT[O_R_Auto] AND $IN[I_SZ2_F_Mot]
  ;Schweissung i.O
  $OUT[O_Kb2_WPS_io]=$OUT[O_R_Auto] AND NOT $FLAG[F_SK2_S_niO]
  ;Schweissung n.i.O
  $OUT[O_Kb2_WP_nio]=$OUT[O_R_Auto] AND $FLAG[F_SK2_S_niO]
  ;Warngrenze verletzt in Folge
  $OUT[O_Kb2_W_Folg]=$OUT[O_R_Auto] AND $IN[I_Kb2_W_Folg]
  ;Phasenueberwachung
  $OUT[O_Kb2_Ph_nio]=$OUT[O_R_Auto] AND $IN[I_Kb2_Ph_nio]
  ;Ueberstrom Primaerseite
  $OUT[O_Kb2_Primae]=$OUT[O_R_Auto] AND $IN[I_Kb2_Primae]
  ;Fehler Stromsensor
  $OUT[O_Kb2_F_Stro]=$OUT[O_R_Auto] AND $IN[I_Kb2_F_Stro]
  ;Fehler Spannungssensor
  $OUT[O_Kb2_F_Span]=$OUT[O_R_Auto] AND $IN[I_Kb2_F_Span]
  ;Überstrom 24 V DC
  $OUT[O_Kb2_24V]=$OUT[O_R_Auto] AND $IN[I_Kb2_24V]
  ;Uebertemperatur Inverter
  $OUT[O_Kb2_Invert]=$OUT[O_R_Auto] AND $IN[I_Kb2_Invert]
  ;Sammelstoerung
  $OUT[O_Kb2_Sammel]=$OUT[O_R_Auto] AND $COULD_START_MOTION AND ($IN[I_Kb2_Sammel] OR $FLAG[F_SZ2_Sammel] OR $FLAG[F_SK2_Sammel] OR SZ_LBitFeh[2]) AND $timer_flag[TimerNr_Ein]
ELSE
  ;Vorwarnung Zange
  $OUT[O_SZ2_W_SZ]=($OUT[O_R_Auto] AND $IN[I_SZ2_W_SZ] OR (Q_T_SZ2_VW>3) OR (Q_T_SZ2_kD>50))
  ;Warnung Schmierung
  $OUT[O_SZ2_W_Schm]=$OUT[O_R_Auto] AND $IN[I_SZ2_W_Schm]
  ;Kraftaufbau zu lange
  $OUT[O_SZ2_F_Kraf]=$OUT[O_R_Auto] AND $IN[I_SZ2_F_Kraf]
  ;Programmfehler/falsche Kraftvorgabe
  $OUT[O_SZ2_F_Prog]=$OUT[O_R_Auto] AND $IN[I_SZ2_F_Prog]
  ;Zielposition ungueltig
  $OUT[O_SZ2_F_Ziel]=$OUT[O_R_Auto] AND $IN[I_SZ2_F_Ziel]
  ;Bauteilfehler
  $OUT[O_SZ2_F_Baut]=$OUT[O_R_Auto] AND $IN[I_SZ2_F_Baut]
  ;Zange geht schwer
  $OUT[O_SZ2_F_schw]=$OUT[O_R_Auto] AND $IN[I_SZ2_F_schw]
  ;Fraesen n.i.O.
  $OUT[O_SZ2_F_Frae]=$OUT[O_R_Auto] AND $IN[I_SZ2_F_Frae]
  ;Fehler Kappenverschleiss/Geometrie
  $OUT[O_SZ2_F_Geom]=$OUT[O_R_Auto] AND ($IN[I_SZ2_F_Kapp] OR $IN[I_SZ2_F_Geom] OR $FLAG[F_SZ2_Kapp])
  ;Fehler Ausgleichssystem
  $OUT[O_SZ2_F_Ausg]=($OUT[O_R_Auto] AND $IN[I_SZ2_F_Ausg] OR (Q_T_SZ2_Fe>3))
  ;Fehler Steuerung/Regler
  $OUT[O_SZ2_F_Steu]=$OUT[O_R_Auto] AND $COULD_START_MOTION AND $IN[I_SZ2_F_Steu]
  ;Fehler Temperatur Motor/Trafo
  $OUT[O_SZ2_F_Temp]=$OUT[O_R_Auto] AND ($IN[I_SZ2_F_Traf] OR $IN[I_SZ2_F_Mot])
  ;Sammelstoerung
  $OUT[O_SZ2_Sammel]=$OUT[O_R_Auto] AND $COULD_START_MOTION AND ($IN[I_SZ2_Sammel] OR $FLAG[F_SZ2_Sammel] OR SZ_LBitFeh[2]) AND $timer_flag[TimerNr_Ein]
ENDIF
;Ausgabe Zangencode
IF Mit_Komb_ST THEN
  Kb2_ZCode=1
ELSE
  EZ2_ZCode=1
ENDIF
;
;FOLD SZ-Tastbetrieb ruecksetzen
IF Mit_Komb_ST2 THEN
  Temp_Komb_2=($OUT[O_Kb2_t_zu] OR $OUT[O_Kb2_t_auf])
ENDIF
IF $OUT[O_R_Hand] AND TAST_AKTIV_2 AND NOT $OUT[O_SZ2_t_auf] AND NOT $OUT[O_SZ2_t_zu] AND NOT Temp_Komb_2 THEN
  TAST_AKTIV_2=FALSE
  $OUT[O_SZ2_FRG]=FALSE
  schleppfehler=TRUE
  sf_prog_status=#user_act
  $OUT[O_SZ2_SPos_g]=FALSE
ENDIF
;ENDFOLD
;
;FOLD SZ INIT Zangenfunktion
IF $OUT[O_R_Hand] AND NOT $OUT[O_R_Auto] AND $COULD_START_MOTION AND ((NOT $OUT[O_R_Proz_akt] AND NOT $OUT[O_R_bewegt]) OR (R1AusgleichFunktion>0)) THEN
  IF Mit_Komb_ST2 THEN
    Temp_Komb_2=$OUT[O_Kb2_t_zu]
  ENDIF
  IF ($OUT[O_SZ2_S_TPos] OR $OUT[O_SZ2_ref] OR $OUT[O_SZ2_auf] OR $OUT[O_SZ2_zu] OR Temp_Komb_2 OR $OUT[O_SZ2_t_auf] OR $OUT[O_SZ2_t_zu] OR $OUT[O_SZ2_Teach] OR $OUT[O_SZ2_D_Auf] OR $OUT[O_SZ2_Du_Zu]) THEN
    CheckZangenFunktion()
    Zangenfunktion()
  ENDIF
ELSE
  IF $OUT[O_SZ2_Teach] OR $OUT[O_SZ2_D_Auf] OR $OUT[O_SZ2_Du_Zu] THEN
    $OUT[O_SZ2_Teach]=FALSE
    $OUT[O_SZ2_D_Auf]=FALSE
    $OUT[O_SZ2_Du_Zu]=FALSE
    S_Zangen_Msg(44,#NotifyMsg)
  ENDIF
ENDIF
;ENDFOLD
;
;FOLD Ruecksetzen Zangenfunktion
IF ($OUT[O_R_Hand] AND ($PRO_MODE1==#BSTEP)) OR ($OUT[O_R_Hand] AND NOT $FLAG[F_SZ_AH_KOMP] AND $OUT[O_R_bewegt] AND (R1AusgleichFunktion==0)) OR ($OUT[O_R_Hand] AND NOT $COULD_START_MOTION AND (HAND_FKT1 OR HAND_FKT2)) THEN
  IF NOT ($OUT[O_SZ2_Re_aus] OR $OUT[O_SZ2_MnFrae] OR $OUT[O_Kb2_MnFrae] OR $FLAG[F_SZ2_FRG_FR]) THEN
    $OUT[O_SZ2_S_TPos]=FALSE
    $OUT[O_SZ2_ref]=FALSE
    $OUT[O_SZ2_FRG]=FALSE
    $OUT[O_SZ2_auf]=FALSE
    $OUT[O_SZ2_zu]=FALSE
    $OUT[O_SZ2_t_auf]=FALSE
    $OUT[O_SZ2_t_zu]=FALSE
    IF Mit_Komb_ST2 THEN
      $OUT[O_Kb2_t_auf]=FALSE
      $OUT[O_Kb2_t_zu]=FALSE
    ENDIF
  ENDIF
  HAND_FKT1=FALSE
  HAND_FKT2=FALSE
ENDIF
;ENDFOLD
;
;FOLD EZ Oeffnungsmass beim Schwenken pruefen
;EZ/SP2
IF ($softplcint[2]>0) AND $OUT[O_SZ2_FRG] AND (Varstate("act_P1")==#initialized) THEN
  IF ($softplcint[2]==8) THEN
    $FLAG[F_SZ2_Oeff_iO]=(act_P1.E2>=$COUNT_I[60])
  ENDIF
  IF ($softplcint[2]==9) THEN
    $FLAG[F_SZ2_Oeff_iO]=(act_P1.E3>=$COUNT_I[60])
  ENDIF
  IF ($softplcint[2]==10) THEN
    $FLAG[F_SZ2_Oeff_iO]=(act_P1.E4>=$COUNT_I[60])
  ENDIF
  IF ($softplcint[2]==11) THEN
    $FLAG[F_SZ2_Oeff_iO]=(act_P1.E5>=$COUNT_I[60])
  ENDIF
  IF ($softplcint[2]==12) THEN
    $FLAG[F_SZ2_Oeff_iO]=(act_P1.E6>=$COUNT_I[60])
  ENDIF
ELSE
  $FLAG[F_SZ2_Oeff_iO]=FALSE
ENDIF
;ENDFOLD
;
;FOLD EZ Position nach Messen und Fraesen pruefen
;EZ/SP2
IF ($softplcint[2]>0) AND $FLAG[F_SZ_Anf_Pos] AND $OUT[O_SZ2_FRG] AND (Varstate("act_P1")==#initialized) THEN
  $FLAG[F_SZ_Anf_Pos]=FALSE
  IF ($softplcint[2]==8)  THEN
    $FLAG[F_SZ2_Pos_iO]=((sig2_istpos>=((act_P1.E2*10)-140)) AND (sig2_istpos<=((act_P1.E2*10)+140)))
  ENDIF
  IF ($softplcint[2]==9) THEN
    $FLAG[F_SZ2_Pos_iO]=((sig2_istpos>=((act_P1.E3*10)-140)) AND (sig2_istpos<=((act_P1.E3*10)+140)))
  ENDIF
  IF ($softplcint[2]==10) THEN
    $FLAG[F_SZ2_Pos_iO]=((sig2_istpos>=((act_P1.E4*10)-140)) AND (sig2_istpos<=((act_P1.E4*10)+140)))
  ENDIF
  IF ($softplcint[2]==11) THEN
    $FLAG[F_SZ2_Pos_iO]=((sig2_istpos>=((act_P1.E5*10)-140)) AND (sig2_istpos<=((act_P1.E5*10)+140)))
  ENDIF
  IF ($softplcint[2]==12) THEN
    $FLAG[F_SZ2_Pos_iO]=((sig2_istpos>=((act_P1.E6*10)-140)) AND (sig2_istpos<=((act_P1.E6*10)+140)))
  ENDIF
ENDIF
;ENDFOLD
;
;FOLD Ruecksetzen Ausgabe max. Kappenverschleiss
IF $OUT[O_SZ2_KW_io] THEN
  B_SK2_M_Stdm = FALSE
  B_SK2_V_Stdm = FALSE
  B_SK2_FRG_Ge = TRUE
ENDIF
;ENDFOLD
;
;FOLD Lebensbit
IF Mit_Komb_ST2 THEN
  L_Bit_Kombi(2)
ELSE
  L_Bit_SZ(2)
ENDIF
;ENDFOLD
;
END
;ENDFOLD
;
;-----------------------------------------------------------
;FOLD LOOP S_Zange 3
GLOBAL DEF SZ3_LOOP( )
;
;SZ 3 Funktionstest ohne Bauteil
IF Mit_Komb_ST3 THEN
  $OUT[O_Kb3_FToBT]=$IN[I_FT_o_BT]
  IF (Prog_Nr_Kb3<99) AND ($FLAG[F_SZ3_FRG_FR] OR $OUT[O_R_Wart] OR $OUT[O_R_WartB]) THEN
    Fzg_Typ_SZ3=0
  ENDIF
ELSE
  $OUT[O_SZ3_FToBT]=$IN[I_FT_o_BT] AND (Prog_Nr_SZ3>98)
  IF (Prog_Nr_SZ3<99) AND ($FLAG[F_SZ3_FRG_FR] OR $OUT[O_R_Wart] OR $OUT[O_R_WartB]) THEN
    Fzg_Typ_SZ3=0
    SK3_Fzg_Typ=0
  ENDIF
ENDIF
;
;SZ 3 Anwahl Energiesparmodus
$OUT[O_SZ3_E_Mode] = (($Brake_Sig==0) AND $timer_flag[TimerNr_E_Mo] AND e_Mode_Hilf2)
;
;FOLD SZ Betriebsarten
;BA-Hand an SZ 3 setzen
IF $OUT[O_R_Hand] AND (NOT $COULD_START_MOTION OR HAND_FKT2) THEN
  $OUT[O_SZ3_R_Hand]=TRUE
  $OUT[O_SZ3_R_Auto]=FALSE
ENDIF
;
;BA-AUTO an SZ 3 setzen
IF $OUT[O_R_Hand] AND NOT HAND_FKT2 AND ($OUT[O_R_Proz_akt] OR $OUT[O_R_bewegt] OR TAST_AKTIV_1 OR TAST_AKTIV_2 OR TAST_AKTIV_3 OR HAND_FKT1) AND (R1AusgleichFunktion==0) OR $OUT[O_R_Auto] THEN
  $OUT[O_SZ3_R_Hand]=FALSE
  $OUT[O_SZ3_R_Auto]=TRUE
ENDIF
;ENDFOLD
;
;SZ 3 mit EK-Verschleisswert
$OUT[O_SZ3_Mit_EK]=TRUE
;
;SZ 3 ohne Kraft
IF $IN[I_SZ3_oh_Kra] THEN
  $OUT[O_SZ3_oh_Kra]=TRUE
ELSE
  $OUT[O_SZ3_oh_Kra]=FALSE
ENDIF
;
;SZ Kraftvorgabe in Hand
IF NOT Mit_Komb_ST3  THEN
  IF $OUT[O_R_Hand] AND $FLAG[F_o_Prozess] THEN
    SZ3_Kraft_Soll = M_Kraft_Soll
  ELSE
    SZ3_Kraft_Soll = SK3_Kraft_Soll
  ENDIF
ENDIF
;
;Kompensation der EK durch Roboter
IF AH_Komp AND NOT $FLAG[F_SZ3_m_Komp] AND NOT Mit_Komb_ST3 THEN
  $OUT[O_SZ3_m_RKom]=TRUE
ELSE
  $OUT[O_SZ3_m_RKom]=FALSE
ENDIF
;
;Quittierung Stoerung
IF Mit_Komb_ST3 THEN
  $OUT[O_Kb3_Fe_Res]=($IN[I_Kb3_Sammel] AND $IN[I_R_Quit_St]) OR (($IN[I_R_Quit_Wei] OR $FLAG[F_SZ_Fe_Res]) AND $IN[I_Kb3_Sammel])
ELSE
  $OUT[O_SZ3_Fe_Res]=($IN[I_SZ3_Sammel] AND $IN[I_R_Quit_St]) OR (($IN[I_R_Quit_Wei] OR $FLAG[F_SZ_Fe_Res]) AND $IN[I_SZ3_Sammel])
ENDIF
;
;Ausgabe Statusmeldungen an BMS
IF Mit_Komb_ST3 THEN
  ;Vorwahl mit Strom
  $OUT[O_Kb3_m_Stro]=NOT $IN[I_Kb3_o_Schw] AND NOT $FLAG[F_o_Prozess]
  ;Start Protokoll
  $OUT[O_Kb3_Protok]=$IN[I_Kb3_Protok]
  ;Vorwarnung Zange
  $OUT[O_Kb3_W_SZ]=($IN[I_SZ3_W_SZ] OR (Q_T_SZ3_VW>3) OR (Q_T_SZ3_kD>50))
  ;Warnung Schmierung
  $OUT[O_Kb3_W_Schm]=$IN[I_SZ3_W_Schm]
  ;Fraesanfrage
  $OUT[O_Kb3_FrAnf]=$OUT[O_R_Auto] AND $IN[I_Kb3_FrAnf]
  ;Vorwarnung Kappenstandzeit
  $OUT[O_Kb3_V_Stdm]=($IN[I_Kb3_V_Stdm] OR B_SK3_V_Stdm)
  ;Maximale Kappenstandzeit
  $OUT[O_Kb3_M_Stdm]=($IN[I_SZ3_F_Geom] OR $IN[I_Kb3_M_Stdm] OR B_SK3_M_Stdm)
  ;Kraftaufbau zu lange
  $OUT[O_Kb3_F_Kraf]=$OUT[O_R_Auto] AND $IN[I_SZ3_F_Kraf]
  ;Punktanwahlfehler
  $OUT[O_Kb3_F_Prog]=$OUT[O_R_Auto] AND $IN[I_SZ3_F_Prog]
  ;Zielposition ungueltig
  $OUT[O_Kb3_F_Ziel]=$OUT[O_R_Auto] AND $IN[I_SZ3_F_Ziel]
  ;Bauteilfehler
  $OUT[O_Kb3_F_Baut]=$OUT[O_R_Auto] AND $IN[I_SZ3_F_Baut]
  ;Zange geht schwer
  $OUT[O_Kb3_F_schw]=$OUT[O_R_Auto] AND $IN[I_SZ3_F_schw]
  ;Fraesen n.i.O.
  $OUT[O_Kb3_F_Frae]=$OUT[O_R_Auto] AND $IN[I_SZ3_F_Frae]
  ;Fehler Kappenverschleiss
  $OUT[O_Kb3_F_KaVe]=$OUT[O_R_Auto] AND $IN[I_SZ3_F_Kapp]
  ;Fehler Geometrie
  $OUT[O_Kb3_F_Geom]=$OUT[O_R_Auto] AND $IN[I_SZ3_F_Geom]
  ;Schleppfehler
  $OUT[O_Kb3_Schlep]=$OUT[O_R_Auto] AND $IN[I_SZ3_F_Schl]
  ;Fehler Ausgleichssystem
  $OUT[O_Kb3_F_Ausg]=$OUT[O_R_Auto] AND ($IN[I_SZ3_F_Ausg] OR (Q_T_SZ3_VW>3))
  ;Fehler Steuerung/Regler
  $OUT[O_Kb3_F_Steu]=$OUT[O_R_Auto] AND $COULD_START_MOTION AND $IN[I_SZ3_F_Steu]
  ;Fehler Temperatur Trafo
  $OUT[O_Kb3_FT_Tra]=$OUT[O_R_Auto] AND $IN[I_SZ3_F_Traf]
  ;Fehler Temperatur Motor
  $OUT[O_Kb3_FT_Mot]=$OUT[O_R_Auto] AND $IN[I_SZ3_F_Mot]
  ;Schweissung i.O
  $OUT[O_Kb3_WPS_io]=$OUT[O_R_Auto] AND NOT $FLAG[F_SK3_S_niO]
  ;Schweissung n.i.O
  $OUT[O_Kb3_WP_nio]=$OUT[O_R_Auto] AND $FLAG[F_SK3_S_niO]
  ;Warngrenze verletzt in Folge
  $OUT[O_Kb3_W_Folg]=$OUT[O_R_Auto] AND $IN[I_Kb3_W_Folg]
  ;Phasenueberwachung
  $OUT[O_Kb3_Ph_nio]=$OUT[O_R_Auto] AND $IN[I_Kb3_Ph_nio]
  ;Ueberstrom Primaerseite
  $OUT[O_Kb3_Primae]=$OUT[O_R_Auto] AND $IN[I_Kb3_Primae]
  ;Fehler Stromsensor
  $OUT[O_Kb3_F_Stro]=$OUT[O_R_Auto] AND $IN[I_Kb3_F_Stro]
  ;Fehler Spannungssensor
  $OUT[O_Kb3_F_Span]=$OUT[O_R_Auto] AND $IN[I_Kb3_F_Span]
  ;Überstrom 24 V DC
  $OUT[O_Kb3_24V]=$OUT[O_R_Auto] AND $IN[I_Kb3_24V]
  ;Uebertemperatur Inverter
  $OUT[O_Kb3_Invert]=$OUT[O_R_Auto] AND $IN[I_Kb3_Invert]
  ;Sammelstoerung
  $OUT[O_Kb3_Sammel]=$OUT[O_R_Auto] AND $COULD_START_MOTION AND ($IN[I_Kb3_Sammel] OR $FLAG[F_SZ3_Sammel] OR $FLAG[F_SK3_Sammel] OR SZ_LBitFeh[3]) AND $timer_flag[TimerNr_Ein]
ELSE
  ;Vorwarnung Zange
  $OUT[O_SZ3_W_SZ]=($OUT[O_R_Auto] AND $IN[I_SZ3_W_SZ] OR (Q_T_SZ3_VW>3) OR (Q_T_SZ3_kD>50))
  ;Warnung Schmierung
  $OUT[O_SZ3_W_Schm]=$OUT[O_R_Auto] AND $IN[I_SZ3_W_Schm]
  ;Kraftaufbau zu lange
  $OUT[O_SZ3_F_Kraf]=$OUT[O_R_Auto] AND $IN[I_SZ3_F_Kraf]
  ;Programmfehler/falsche Kraftvorgabe
  $OUT[O_SZ3_F_Prog]=$OUT[O_R_Auto] AND $IN[I_SZ3_F_Prog]
  ;Zielposition ungueltig
  $OUT[O_SZ3_F_Ziel]=$OUT[O_R_Auto] AND $IN[I_SZ3_F_Ziel]
  ;Bauteilfehler
  $OUT[O_SZ3_F_Baut]=$OUT[O_R_Auto] AND $IN[I_SZ3_F_Baut]
  ;Zange geht schwer
  $OUT[O_SZ3_F_schw]=$OUT[O_R_Auto] AND $IN[I_SZ3_F_schw]
  ;Fraesen n.i.O.
  $OUT[O_SZ3_F_Frae]=$OUT[O_R_Auto] AND $IN[I_SZ3_F_Frae]
  ;Fehler Kappenverschleiss/Geometrie
  $OUT[O_SZ3_F_Geom]=$OUT[O_R_Auto] AND ($IN[I_SZ3_F_Kapp] OR $IN[I_SZ3_F_Geom] OR $FLAG[F_SZ3_Kapp])
  ;Fehler Ausgleichssystem
  $OUT[O_SZ3_F_Ausg]=($OUT[O_R_Auto] AND $IN[I_SZ3_F_Ausg] OR (Q_T_SZ3_Fe>3))
  ;Fehler Steuerung/Regler
  $OUT[O_SZ3_F_Steu]=$OUT[O_R_Auto] AND $COULD_START_MOTION AND $IN[I_SZ3_F_Steu]
  ;Fehler Temperatur Motor/Trafo
  $OUT[O_SZ3_F_Temp]=$OUT[O_R_Auto] AND ($IN[I_SZ3_F_Traf] OR $IN[I_SZ3_F_Mot])
  ;Sammelstoerung
  $OUT[O_SZ3_Sammel]=$OUT[O_R_Auto] AND $COULD_START_MOTION AND ($IN[I_SZ3_Sammel] OR $FLAG[F_SZ3_Sammel] OR SZ_LBitFeh[3]) AND $timer_flag[TimerNr_Ein]
ENDIF
;Ausgabe Zangencode
IF Mit_Komb_ST THEN
  Kb3_ZCode=1
ELSE
  EZ3_ZCode=1
ENDIF
;
;FOLD SZ-Tastbetrieb ruecksetzen
IF Mit_Komb_ST3 THEN
  Temp_Komb_3=($OUT[O_Kb3_t_zu] OR $OUT[O_Kb3_t_auf])
ENDIF
IF $OUT[O_R_Hand] AND TAST_AKTIV_3 AND NOT $OUT[O_SZ3_t_auf] AND NOT $OUT[O_SZ3_t_zu] AND NOT Temp_Komb_3 THEN
  TAST_AKTIV_3=FALSE
  $OUT[O_SZ3_FRG]=FALSE
  schleppfehler=TRUE
  sf_prog_status=#user_act
  $OUT[O_SZ3_SPos_g]=FALSE
ENDIF
;ENDFOLD
;
;FOLD SZ INIT Zangenfunktion
IF $OUT[O_R_Hand] AND NOT $OUT[O_R_Auto] AND $COULD_START_MOTION AND ((NOT $OUT[O_R_Proz_akt] AND NOT $OUT[O_R_bewegt]) OR (R1AusgleichFunktion>0)) THEN
  IF Mit_Komb_ST3 THEN
    Temp_Komb_3=$OUT[O_Kb3_t_zu]
  ENDIF
  IF ($OUT[O_SZ3_S_TPos] OR $OUT[O_SZ3_ref] OR $OUT[O_SZ3_auf] OR $OUT[O_SZ3_zu] OR Temp_Komb_3 OR $OUT[O_SZ3_t_auf] OR $OUT[O_SZ3_t_zu] OR $OUT[O_SZ3_Teach] OR $OUT[O_SZ3_D_Auf] OR $OUT[O_SZ3_Du_Zu]) THEN
    CheckZangenFunktion()
    Zangenfunktion()
  ENDIF
ELSE
  IF $OUT[O_SZ3_Teach] OR $OUT[O_SZ3_D_Auf] OR $OUT[O_SZ3_Du_Zu] THEN
    $OUT[O_SZ3_Teach]=FALSE
    $OUT[O_SZ3_D_Auf]=FALSE
    $OUT[O_SZ3_Du_Zu]=FALSE
    S_Zangen_Msg(54,#NotifyMsg)
  ENDIF
ENDIF
;ENDFOLD
;
;FOLD Ruecksetzen Zangenfunktion
IF ($OUT[O_R_Hand] AND ($PRO_MODE1==#BSTEP)) OR ($OUT[O_R_Hand] AND NOT $FLAG[F_SZ_AH_KOMP] AND $OUT[O_R_bewegt] AND (R1AusgleichFunktion==0)) OR ($OUT[O_R_Hand] AND NOT $COULD_START_MOTION AND (HAND_FKT1 OR HAND_FKT2)) THEN
  IF NOT ($OUT[O_SZ3_Re_aus] OR $OUT[O_SZ3_MnFrae] OR $OUT[O_Kb3_MnFrae] OR $FLAG[F_SZ3_FRG_FR]) THEN
    $OUT[O_SZ3_S_TPos]=FALSE
    $OUT[O_SZ3_ref]=FALSE
    $OUT[O_SZ3_FRG]=FALSE
    $OUT[O_SZ3_auf]=FALSE
    $OUT[O_SZ3_zu]=FALSE
    $OUT[O_SZ3_t_auf]=FALSE
    $OUT[O_SZ3_t_zu]=FALSE
    IF Mit_Komb_ST3 THEN
      $OUT[O_Kb3_t_auf]=FALSE
      $OUT[O_Kb3_t_zu]=FALSE
    ENDIF
  ENDIF
  HAND_FKT1=FALSE
  HAND_FKT2=FALSE
ENDIF
;ENDFOLD
;
;FOLD EZ Oeffnungsmass beim Schwenken pruefen
;EZ/SP3
IF ($softplcint[3]>0) AND $OUT[O_SZ3_FRG] AND (Varstate("act_P1")==#initialized) THEN
  IF ($softplcint[3]==8) THEN
    $FLAG[F_SZ3_Oeff_iO]=(act_P1.E2>=$COUNT_I[60])
  ENDIF
  IF ($softplcint[3]==9) THEN
    $FLAG[F_SZ3_Oeff_iO]=(act_P1.E3>=$COUNT_I[60])
  ENDIF
  IF ($softplcint[3]==10) THEN
    $FLAG[F_SZ3_Oeff_iO]=(act_P1.E4>=$COUNT_I[60])
  ENDIF
  IF ($softplcint[3]==11) THEN
    $FLAG[F_SZ3_Oeff_iO]=(act_P1.E5>=$COUNT_I[60])
  ENDIF
  IF ($softplcint[3]==12) THEN
    $FLAG[F_SZ3_Oeff_iO]=(act_P1.E6>=$COUNT_I[60])
  ENDIF
ELSE
  $FLAG[F_SZ3_Oeff_iO]=FALSE
ENDIF
;ENDFOLD
;
;FOLD EZ Position nach Messen und Fraesen pruefen
;EZ/SP3
IF ($softplcint[3]>0) AND $FLAG[F_SZ_Anf_Pos] AND $OUT[O_SZ3_FRG] AND (Varstate("act_P1")==#initialized) THEN
  $FLAG[F_SZ_Anf_Pos]=FALSE
  IF ($softplcint[3]==8) THEN
    $FLAG[F_SZ3_Pos_iO] = ((sig3_istpos>=((act_P1.E2*10)-140)) AND (sig3_istpos<=((act_P1.E2*10)+140)))
  ENDIF
  IF ($softplcint[3]==9) THEN
    $FLAG[F_SZ3_Pos_iO] = ((sig3_istpos>=((act_P1.E3*10)-140)) AND (sig3_istpos<=((act_P1.E3*10)+140)))
  ENDIF
  IF ($softplcint[3]==10) THEN
    $FLAG[F_SZ3_Pos_iO] = ((sig3_istpos>=((act_P1.E4*10)-140)) AND (sig3_istpos<=((act_P1.E4*10)+140)))
  ENDIF
  IF ($softplcint[3]==11) THEN
    $FLAG[F_SZ3_Pos_iO] = ((sig3_istpos>=((act_P1.E5*10)-140)) AND (sig3_istpos<=((act_P1.E5*10)+140)))
  ENDIF
  IF ($softplcint[3]==12) THEN
    $FLAG[F_SZ3_Pos_iO] = ((sig3_istpos>=((act_P1.E6*10)-140)) AND (sig3_istpos<=((act_P1.E6*10)+140)))
  ENDIF
ENDIF
;ENDFOLD
;
;FOLD Ruecksetzen Ausgabe max. Kappenverschleiss
IF $OUT[O_SZ3_KW_io] THEN
  B_SK3_M_Stdm = FALSE
  B_SK3_V_Stdm = FALSE
  B_SK3_FRG_Ge = TRUE
ENDIF
;ENDFOLD
;
;FOLD Lebensbit
IF Mit_Komb_ST3 THEN
  L_Bit_Kombi(3)
ELSE
  L_Bit_SZ(3)
ENDIF
;ENDFOLD
;
END
;ENDFOLD
;
;------------------------------------------------------
;FOLD Zangenfunktion
DEF CheckZangenfunktion()
IF ($Pro_state1 == #P_Free) THEN
  IF $OUT[O_SZ1_Teach] OR $OUT[O_SZ1_D_Auf] OR $OUT[O_SZ1_Du_Zu] THEN
    $OUT[O_SZ1_Teach]=FALSE
    $OUT[O_SZ1_D_Auf]=FALSE
    $OUT[O_SZ1_Du_Zu]=FALSE
    S_Zangen_Msg(21,#NotifyMsg)
  ENDIF
  IF $OUT[O_SZ2_Teach] OR $OUT[O_SZ2_D_Auf] OR $OUT[O_SZ2_Du_Zu] THEN
    $OUT[O_SZ2_Teach]=FALSE
    $OUT[O_SZ2_D_Auf]=FALSE
    $OUT[O_SZ2_Du_Zu]=FALSE
    S_Zangen_Msg(21,#NotifyMsg)
  ENDIF
  IF $OUT[O_SZ3_Teach] OR $OUT[O_SZ3_D_Auf] OR $OUT[O_SZ3_Du_Zu] THEN
    $OUT[O_SZ3_Teach]=FALSE
    $OUT[O_SZ3_D_Auf]=FALSE
    $OUT[O_SZ3_Du_Zu]=FALSE
    S_Zangen_Msg(21,#NotifyMsg)
  ENDIF
  RETURN
ENDIF
IF ($Pro_state1 == #P_Reset) THEN
  IF $OUT[O_SZ1_Teach] OR $OUT[O_SZ1_D_Auf] OR $OUT[O_SZ1_Du_Zu] THEN
    $OUT[O_SZ1_Teach]=FALSE
    $OUT[O_SZ1_D_Auf]=FALSE
    $OUT[O_SZ1_Du_Zu]=FALSE
    S_Zangen_Msg(22,#NotifyMsg)
  ENDIF
  IF $OUT[O_SZ2_Teach] OR $OUT[O_SZ2_D_Auf] OR $OUT[O_SZ2_Du_Zu] THEN
    $OUT[O_SZ2_Teach]=FALSE
    $OUT[O_SZ2_D_Auf]=FALSE
    $OUT[O_SZ2_Du_Zu]=FALSE
    S_Zangen_Msg(22,#NotifyMsg)
  ENDIF
  IF $OUT[O_SZ3_Teach] OR $OUT[O_SZ3_D_Auf] OR $OUT[O_SZ3_Du_Zu] THEN
    $OUT[O_SZ3_Teach]=FALSE
    $OUT[O_SZ3_D_Auf]=FALSE
    $OUT[O_SZ3_Du_Zu]=FALSE
    S_Zangen_Msg(22,#NotifyMsg)
  ENDIF
  RETURN
ENDIF
IF NOT($ON_Path) THEN
  IF $OUT[O_SZ1_Teach] OR $OUT[O_SZ1_D_Auf] OR $OUT[O_SZ1_Du_Zu] THEN
    $OUT[O_SZ1_Teach]=FALSE
    $OUT[O_SZ1_D_Auf]=FALSE
    $OUT[O_SZ1_Du_Zu]=FALSE
    S_Zangen_Msg(24,#NotifyMsg)
  ENDIF
  IF $OUT[O_SZ2_Teach] OR $OUT[O_SZ2_D_Auf] OR $OUT[O_SZ2_Du_Zu] THEN
    $OUT[O_SZ2_Teach]=FALSE
    $OUT[O_SZ2_D_Auf]=FALSE
    $OUT[O_SZ2_Du_Zu]=FALSE
    S_Zangen_Msg(24,#NotifyMsg)
  ENDIF
  IF $OUT[O_SZ3_Teach] OR $OUT[O_SZ3_D_Auf] OR $OUT[O_SZ3_Du_Zu] THEN
    $OUT[O_SZ3_Teach]=FALSE
    $OUT[O_SZ3_D_Auf]=FALSE
    $OUT[O_SZ3_Du_Zu]=FALSE
    S_Zangen_Msg(24,#NotifyMsg)
  ENDIF
ENDIF
IF $OUT[O_SZ1_Teach]  and ($FLAG[F_o_Ausgl]) THEN
  ; teach funktion nicht wenn kein SStep
  $OUT[O_SZ1_Teach]=FALSE
  $OUT[O_SZ1_S_Tpos]=truE
  ;SyncMoveMessage(39,#NotifyMsg)
  RETURN
ENDIF
IF $OUT[O_SZ2_Teach]  and ($FLAG[F_o_Ausgl]) THEN
  ; teach funktion nicht wenn kein SStep
  $OUT[O_SZ2_Teach]=FALSE
  $OUT[O_SZ2_S_Tpos]=truE
  ;SyncMoveMessage(39,#NotifyMsg)
  RETURN
ENDIF
IF $OUT[O_SZ3_Teach]  and ($FLAG[F_o_Ausgl]) THEN
  ; teach funktion nicht wenn kein SStep
  $OUT[O_SZ3_Teach]=FALSE
  $OUT[O_SZ3_S_Tpos]=truE
  ;SyncMoveMessage(39,#NotifyMsg)
  RETURN
ENDIF
IF $OUT[O_SZ1_Teach]  and ($Pro_mode1<>#MSTEP) THEN
  ; teach funktion nicht wenn kein SStep
  $OUT[O_SZ1_Teach]=FALSE
  S_Zangen_Msg(23,#NotifyMsg)
  RETURN
ENDIF
IF $OUT[O_SZ2_Teach] and ($Pro_mode1<>#MSTEP) THEN
  ; teach funktion nicht wenn kein SStep
  $OUT[O_SZ2_Teach]=FALSE
  S_Zangen_Msg(23,#NotifyMsg)
  RETURN
ENDIF
IF $OUT[O_SZ3_Teach] and ($Pro_mode1<>#MSTEP) THEN
  ; teach funktion nicht wenn kein SStep
  $OUT[O_SZ3_Teach]=FALSE
  S_Zangen_Msg(23,#NotifyMsg)
  RETURN
ENDIF
IF $OUT[O_SZ1_Du_Zu]  and ($FLAG[F_o_Ausgl]) THEN
  ; teach funktion nicht wenn kein Flag [F_o_Ausgl]
  $OUT[O_SZ1_Du_Zu]=FALSE
  $OUT[O_SZ1_Zu]=truE
  ;SyncMoveMessage(80,#NotifyMsg)
  RETURN
ENDIF
IF $OUT[O_SZ1_D_auf]  and ($FLAG[F_o_Ausgl]) THEN
  ; teach funktion nicht wenn kein Flag [F_o_Ausgl]
  $OUT[O_SZ1_D_auf]=FALSE
  $OUT[O_SZ1_auf]=truE
  ;SyncMoveMessage(80,#NotifyMsg)
  RETURN
ENDIF

IF R1AusgleichFunktion==0 THEN
  IF $OUT[O_SZ1_Teach] then
    ;teachen SZ1 EIN
	;xxxxxxxxxx   flegel  xxxxx
     if ($mode_op==#t1) and ($ov_pro<>50) then
      ov_merk=$ov_pro
      $ov_pro=50
     endif
     if ($mode_op==#t2) and ($ov_pro<>5) then
      ov_merk=$ov_pro
      $ov_pro=5
     endif
    R1AusgleichFunktion=1
    $OUT[O_SZ1_Teach]=FALSE
    S_Zangen_Msg(31,#NotifyMsg)
  ENDIF
  IF $OUT[O_SZ1_D_Auf] then
    ;Oeffen SZ1
    R1AusgleichFunktion=2
    $OUT[O_SZ1_D_Auf]=FALSE
    S_Zangen_Msg(32,#NotifyMsg)
  ENDIF
  IF $OUT[O_SZ1_Du_Zu] then
    ;schliessen SZ1 EIN
    R1AusgleichFunktion=3
    $OUT[O_SZ1_Du_Zu]=FALSE
    S_Zangen_Msg(33,#NotifyMsg)
  ENDIF
  IF $OUT[O_SZ2_Teach] then
    ;teachen SZ2 EIN
	;xxxxxxxxxx   flegel  xxxxx
     if ($mode_op==#t1) and ($ov_pro<>50) then
      ov_merk=$ov_pro
      $ov_pro=50
     endif
     if ($mode_op==#t2) and ($ov_pro<>5) then
      ov_merk=$ov_pro
      $ov_pro=5
     endif
    R1AusgleichFunktion=11
    $OUT[O_SZ2_Teach]=FALSE
    S_Zangen_Msg(41,#NotifyMsg)
  ENDIF
IF $OUT[O_SZ2_Du_Zu]  and ($FLAG[F_o_Ausgl]) THEN
  ; teach funktion nicht wenn kein Flag [F_o_Ausgl]
  $OUT[O_SZ2_Du_Zu]=FALSE
  $OUT[O_SZ2_Zu]=truE
  ;SyncMoveMessage(80,#NotifyMsg)
  RETURN
ENDIF
IF $OUT[O_SZ2_D_auf]  and ($FLAG[F_o_Ausgl]) THEN
  ; teach funktion nicht wenn kein Flag [F_o_Ausgl]
  $OUT[O_SZ2_D_auf]=FALSE
  $OUT[O_SZ2_auf]=truE
  ;SyncMoveMessage(80,#NotifyMsg)
  RETURN
ENDIF

  IF $OUT[O_SZ2_D_Auf] then
    ;Oeffen SZ2
    R1AusgleichFunktion=12
    $OUT[O_SZ2_D_Auf]=FALSE
    S_Zangen_Msg(42,#NotifyMsg)
  ENDIF
  IF $OUT[O_SZ2_Du_Zu] then
    ;schliessen SZ2 EIN
    R1AusgleichFunktion=13
    $OUT[O_SZ2_Du_Zu]=FALSE
    S_Zangen_Msg(43,#NotifyMsg)
  ENDIF
  IF $OUT[O_SZ3_Teach] then
    ;teachen SZ3 EIN
	;xxxxxxxxxx   flegel  xxxxx
     if ($mode_op==#t1) and ($ov_pro<>50) then
      ov_merk=$ov_pro
      $ov_pro=50
     endif
     if ($mode_op==#t2) and ($ov_pro<>5) then
      ov_merk=$ov_pro
      $ov_pro=5
     endif
    R1AusgleichFunktion=21
    $OUT[O_SZ3_Teach]=FALSE
    S_Zangen_Msg(51,#NotifyMsg)
  ENDIF
IF $OUT[O_SZ3_Du_Zu]  and ($FLAG[F_o_Ausgl]) THEN
  ; teach funktion nicht wenn kein Flag [F_o_Ausgl]
  $OUT[O_SZ3_Du_Zu]=FALSE
  $OUT[O_SZ3_Zu]=truE
  ;SyncMoveMessage(80,#NotifyMsg)
  RETURN
ENDIF
IF $OUT[O_SZ3_D_auf]  and ($FLAG[F_o_Ausgl]) THEN
  ; teach funktion nicht wenn kein Flag [F_o_Ausgl]
  $OUT[O_SZ3_D_auf]=FALSE
  $OUT[O_SZ3_auf]=truE
  ;SyncMoveMessage(80,#NotifyMsg)
  RETURN
ENDIF

  IF $OUT[O_SZ3_D_Auf] then
    ;Oeffen SZ3
    R1AusgleichFunktion=22
    $OUT[O_SZ3_D_Auf]=FALSE
    S_Zangen_Msg(52,#NotifyMsg)
  ENDIF
  IF $OUT[O_SZ3_Du_Zu] then
    ;schliessen SZ3 EIN
    R1AusgleichFunktion=23
    $OUT[O_SZ3_Du_Zu]=FALSE
    S_Zangen_Msg(53,#NotifyMsg)
  ENDIF
ELSE
  IF $OUT[O_SZ1_Teach] OR $OUT[O_SZ1_D_Auf] OR $OUT[O_SZ1_Du_Zu] THEN
    S_Zangen_Msg(35,#NotifyMsg); Zangenfunktion bereits aktiv
    $OUT[O_SZ1_Teach]=FALSE
    $OUT[O_SZ1_D_Auf]=FALSE
    $OUT[O_SZ1_Du_Zu]=FALSE
  ENDIF
  IF $OUT[O_SZ2_Teach] OR $OUT[O_SZ2_D_Auf] OR $OUT[O_SZ2_Du_Zu] THEN
    S_Zangen_Msg(45,#NotifyMsg); Zangenfunktion bereits aktiv
    $OUT[O_SZ2_Teach]=FALSE
    $OUT[O_SZ2_D_Auf]=FALSE
    $OUT[O_SZ2_Du_Zu]=FALSE
  ENDIF
  IF $OUT[O_SZ3_Teach] OR $OUT[O_SZ3_D_Auf] OR $OUT[O_SZ3_Du_Zu] THEN
    S_Zangen_Msg(55,#NotifyMsg); Zangenfunktion bereits aktiv
    $OUT[O_SZ3_Teach]=FALSE
    $OUT[O_SZ3_D_Auf]=FALSE
    $OUT[O_SZ3_Du_Zu]=FALSE
  ENDIF
ENDIF
END
;
;------------------------------------------------------
DEF Zangenfunktion()
;Schweisszangen
;SZ 1 Oeffnen in Hand
IF $OUT[O_SZ1_auf] THEN
  $OUT[O_SZ1_FRG]=TRUE
  $OUT[O_SZ1_zu]=FALSE
  $OUT[O_Kb1_zu_o_S]=FALSE
  HAND_FKT1=TRUE
  IF $IN[I_SZ1_auf] THEN
    $OUT[O_SZ1_auf]=FALSE
  ENDIF
ENDIF
;
;SZ 1 Schliessen in Hand
IF Mit_Komb_ST1 THEN
  IF $OUT[O_Kb1_zu_o_S] THEN
    $OUT[O_SZ1_FRG]=TRUE
    $OUT[O_SZ1_auf]=FALSE
    HAND_FKT1=TRUE
    IF $IN[I_SZ1_zu] THEN
      $OUT[O_Kb1_zu_o_S]=FALSE
    ENDIF
  ENDIF
ELSE
  IF $OUT[O_SZ1_zu] THEN
    $OUT[O_SZ1_FRG]=TRUE
    $OUT[O_SZ1_auf]=FALSE
    HAND_FKT1=TRUE
    IF $IN[I_SZ1_zu] THEN
      $OUT[O_SZ1_zu]=FALSE
    ENDIF
  ENDIF
ENDIF
;
; ~~~~~~~~~~~~ VW Teil-Anfang~~~~~~~~
;SZ 1 Fahrt auf Teachposition ausloesen
IF Mit_Komb_ST THEN
	IF $OUT[O_SZ1_S_TPos] THEN
		$OUT[O_SZ1_TPos_u]=FALSE
		TeachPos=FALSE
		HAND_FKT2=TRUE
		WAIT SEC 0.4
		$OUT[O_SZ1_FRG]=TRUE
		IF $IN[I_SZ1_TPos_g] THEN
			TeachPos=TRUE
			$OUT[O_SZ1_S_TPos]=FALSE
			$OUT[O_SZ1_TPos_u]=TRUE
			sf_prog_status=#user_act
			$OUT[O_SZ1_SPos_g]=FALSE
			WAIT SEC 0.4
			schleppfehler=TRUE
			WAIT SEC 1.0
       IF  (schleppfehler==FALSE) THEN
				$OUT[O_SZ1_FRG]=FALSE
				$OUT[O_SZ1_TPos_u]=FALSE
				HAND_FKT2=FALSE
		ENDIF
	ENDIF
   ENDIF
ELSE
   IF $OUT[O_SZ1_S_TPos] THEN
     $OUT[O_SZ1_TPos_u]=FALSE
     TeachPos=FALSE
     HAND_FKT2=TRUE
     WAIT SEC 0.4
     $OUT[O_SZ1_FRG]=TRUE
     IF $IN[I_SZ1_TPos_g] THEN
       TeachPos=TRUE
       $OUT[O_SZ1_S_TPos]=FALSE
       $OUT[O_SZ1_TPos_u]=TRUE
       sf_prog_status=#user_act
       $OUT[O_SZ1_SPos_g]=FALSE
       WAIT SEC 0.4
       schleppfehler=TRUE
       $OUT[O_SZ1_FRG]=FALSE
       $OUT[O_SZ1_TPos_u]=FALSE
       HAND_FKT2=FALSE
     ENDIF
   ENDIF
ENDIF
;
;~~~~~~~~~~~~~~~VW-Teil-Ende~~~~~~~~
;
;SZ 1 Referenzieren
IF $OUT[O_SZ1_ref] THEN
  $OUT[O_SZ1_FRG]=TRUE
  HAND_FKT2=TRUE
  IF NOT $IN[I_SZ1_ref] THEN
    B_SZ1_n_Ref=TRUE
  ENDIF
  IF $IN[I_SZ1_ref] AND $IN[I_SZ1_IPos_g] AND B_SZ1_n_Ref THEN
    $OUT[O_SZ1_ref]=FALSE
    $OUT[O_SZ1_FRG]=FALSE
    HAND_FKT2=FALSE
	 B_SZ1_n_Ref=FALSE
    S_Zangen_Msg(1,#NotifyMsg)
  ENDIF
ENDIF
;
;SZ 1 Tastend Auf
IF Mit_Komb_ST1 THEN
  IF $OUT[O_Kb1_t_auf] THEN
    TAST_AKTIV_1=TRUE
    $OUT[O_SZ1_FRG]=TRUE
  ENDIF
ELSE
  IF $OUT[O_SZ1_t_auf] THEN
    TAST_AKTIV_1=TRUE
    $OUT[O_SZ1_FRG]=TRUE
  ENDIF
ENDIF
;
;SZ 1 Tastend Zu
IF Mit_Komb_ST1 THEN
  IF $OUT[O_Kb1_t_zu] THEN
    TAST_AKTIV_1=TRUE
    $OUT[O_SZ1_FRG]=TRUE
  ENDIF
ELSE
  IF $OUT[O_SZ1_t_zu] THEN
    TAST_AKTIV_1=TRUE
    $OUT[O_SZ1_FRG]=TRUE
  ENDIF
ENDIF
;
;SZ 2 Oeffnen in Hand
IF $OUT[O_SZ2_auf] THEN
  $OUT[O_SZ2_FRG]=TRUE
  $OUT[O_SZ2_zu]=FALSE
  $OUT[O_Kb2_zu_o_S]=FALSE
  HAND_FKT1=TRUE
  IF $IN[I_SZ2_auf] THEN
    $OUT[O_SZ2_auf]=FALSE
  ENDIF
ENDIF
;
;SZ 2 Schliessen in Hand
IF Mit_Komb_ST2 THEN
  IF $OUT[O_Kb2_zu_o_S] THEN
    $OUT[O_SZ2_FRG]=TRUE
    $OUT[O_SZ2_auf]=FALSE
    HAND_FKT1=TRUE
    IF $IN[I_SZ2_zu] THEN
      $OUT[O_Kb2_zu_o_S]=FALSE
    ENDIF
  ENDIF
ELSE
  IF $OUT[O_SZ2_zu] THEN
    $OUT[O_SZ2_FRG]=TRUE
    $OUT[O_SZ2_auf]=FALSE
    HAND_FKT1=TRUE
    IF $IN[I_SZ2_zu] THEN
      $OUT[O_SZ2_zu]=FALSE
    ENDIF
  ENDIF
ENDIF
;
;SZ 2 Fahrt auf Teachposition ausloesen
IF $OUT[O_SZ2_S_TPos] THEN
  $OUT[O_SZ2_TPos_u]=FALSE
  TeachPos=FALSE
  HAND_FKT2=TRUE
  WAIT SEC 0.4
  $OUT[O_SZ2_FRG]=TRUE
  IF $IN[I_SZ2_TPos_g] THEN
    TeachPos=TRUE
    $OUT[O_SZ2_S_TPos]=FALSE
    $OUT[O_SZ2_TPos_u]=TRUE
    sf_prog_status=#user_act
    $OUT[O_SZ2_SPos_g]=FALSE
    schleppfehler=TRUE
    WAIT SEC 0.4
    $OUT[O_SZ2_FRG]=FALSE
    $OUT[O_SZ2_TPos_u]=FALSE
    HAND_FKT2=FALSE
  ENDIF
ENDIF
;
;SZ 2 Referenzieren
IF $OUT[O_SZ2_ref] THEN
  $OUT[O_SZ2_FRG]=TRUE
  HAND_FKT2=TRUE
  IF NOT $IN[I_SZ2_ref] THEN
    B_SZ2_n_Ref=TRUE
  ENDIF
  IF $IN[I_SZ2_ref] AND $IN[I_SZ2_IPos_g] AND B_SZ2_n_Ref THEN
    $OUT[O_SZ2_ref]=FALSE
    $OUT[O_SZ2_FRG]=FALSE
    HAND_FKT2=FALSE
	 B_SZ2_n_Ref=FALSE
    S_Zangen_Msg(2,#NotifyMsg)
  ENDIF
ENDIF
;
;SZ 2 Tastend Auf
IF Mit_Komb_ST2 THEN
  IF $OUT[O_Kb2_t_auf] THEN
    TAST_AKTIV_2=TRUE
    $OUT[O_SZ2_FRG]=TRUE
  ENDIF
ELSE
  IF $OUT[O_SZ2_t_auf] THEN
    TAST_AKTIV_2=TRUE
    $OUT[O_SZ2_FRG]=TRUE
  ENDIF
ENDIF
;
;SZ 2 Tastend Zu
IF Mit_Komb_ST2 THEN
  IF $OUT[O_Kb2_t_zu] THEN
    TAST_AKTIV_2=TRUE
    $OUT[O_SZ2_FRG]=TRUE
  ENDIF
ELSE
  IF $OUT[O_SZ2_t_zu] THEN
    TAST_AKTIV_2=TRUE
    $OUT[O_SZ2_FRG]=TRUE
  ENDIF
ENDIF
;
;SZ 3 Oeffnen in Hand
IF $OUT[O_SZ3_auf] THEN
  $OUT[O_SZ3_FRG]=TRUE
  $OUT[O_SZ3_zu]=FALSE
  $OUT[O_Kb3_zu_o_S]=FALSE
  HAND_FKT1=TRUE
  IF $IN[I_SZ3_auf] THEN
    $OUT[O_SZ3_auf]=FALSE
  ENDIF
ENDIF
;
;SZ 3 Schliessen in Hand
IF Mit_Komb_ST3 THEN
  IF $OUT[O_Kb3_zu_o_S] THEN
    $OUT[O_SZ3_FRG]=TRUE
    $OUT[O_SZ3_auf]=FALSE
    HAND_FKT1=TRUE
    IF $IN[I_SZ3_zu] THEN
      $OUT[O_Kb3_zu_o_S]=FALSE
    ENDIF
  ENDIF
ELSE
  IF $OUT[O_SZ3_zu] THEN
    $OUT[O_SZ3_FRG]=TRUE
    $OUT[O_SZ3_auf]=FALSE
    HAND_FKT1=TRUE
    IF $IN[I_SZ3_zu] THEN
      $OUT[O_SZ3_zu]=FALSE
    ENDIF
  ENDIF
ENDIF
;
;SZ 3 Fahrt auf Teachposition ausloesen
IF $OUT[O_SZ3_S_TPos] THEN
  $OUT[O_SZ3_TPos_u]=FALSE
  TeachPos=FALSE
  HAND_FKT2=TRUE
  WAIT SEC 0.4
  $OUT[O_SZ3_FRG]=TRUE
  IF $IN[I_SZ3_TPos_g] THEN
    TeachPos=TRUE
    $OUT[O_SZ3_S_TPos]=FALSE
    $OUT[O_SZ3_TPos_u]=TRUE
    sf_prog_status=#user_act
    $OUT[O_SZ3_SPos_g]=FALSE
    schleppfehler=TRUE
    WAIT SEC 0.4
    $OUT[O_SZ3_FRG]=FALSE
    $OUT[O_SZ3_TPos_u]=FALSE
    HAND_FKT2=FALSE
  ENDIF
ENDIF
;
;SZ 3 Referenzieren
IF $OUT[O_SZ3_ref] THEN
  $OUT[O_SZ3_FRG]=TRUE
  HAND_FKT2=TRUE
  IF NOT $IN[I_SZ3_ref] THEN
    B_SZ3_n_Ref=TRUE
  ENDIF
  IF $IN[I_SZ3_ref] AND $IN[I_SZ3_IPos_g] AND B_SZ3_n_Ref THEN
    $OUT[O_SZ3_ref]=FALSE
    $OUT[O_SZ3_FRG]=FALSE
    HAND_FKT2=FALSE
	B_SZ3_n_Ref=FALSE
    S_Zangen_Msg(3,#NotifyMsg)
  ENDIF
ENDIF
;
;SZ 3 Tastend Auf
IF Mit_Komb_ST3 THEN
  IF $OUT[O_Kb3_t_auf] THEN
    TAST_AKTIV_3=TRUE
    $OUT[O_SZ3_FRG]=TRUE
  ENDIF
ELSE
  IF $OUT[O_SZ3_t_auf] THEN
    TAST_AKTIV_3=TRUE
    $OUT[O_SZ3_FRG]=TRUE
  ENDIF
ENDIF
;
;SZ 3 Tastend Zu
IF Mit_Komb_ST3 THEN
  IF $OUT[O_Kb3_t_zu] THEN
    TAST_AKTIV_3=TRUE
    $OUT[O_SZ3_FRG]=TRUE
  ENDIF
ELSE
  IF $OUT[O_SZ3_t_zu] THEN
    TAST_AKTIV_3=TRUE
    $OUT[O_SZ3_FRG]=TRUE
  ENDIF
ENDIF
;
END
;ENDFOLD (Zangenfunktion)
;
;~~~~~~~~~VW-Teil-Anfang~~~~~~~~
;
;FOLD LOOP Mutterbuckeln VW-V3
GLOBAL DEF BM1_LOOP( )
  IF $FLAG[F_m_BM1_Einz] OR $FLAG[F_m_BM1_Dopp] THEN
    MIT_BM1=TRUE
  ELSE
    MIT_BM1=FALSE
  ENDIF
;
  ;Ausgabe Fehlermeldungen
  IF MIT_BM1 THEN
   ;
   ;Sammelstoerung
    $OUT[O_BM1_Sammel]=$OUT[O_R_Auto] AND $COULD_START_MOTION AND ($OUT[O_SK1_Sammel] OR $FLAG[F_SK1_Sammel]) AND $timer_flag[TimerNr_Ein]
  ENDIF
;
  IF ($OUT[O_R_Hand] AND NOT $OUT[O_R_Auto] AND $OUT[O_R_RK100] AND NOT $OUT[O_R_Proz_akt] AND NOT $FLAG[F_R_RobMove]) THEN
    ;
    ;BM1 schliessen in Hand ohne Zustellhub
    IF (($OUT[O_BM1_zu]) AND $FLAG[F_m_BM1_Einz] AND NOT $FLAG[F_m_BM1_Dopp] AND NOT $FLAG[F_m_BM2_Einz] AND NOT $FLAG[F_m_BM2_Dopp]) THEN
      SK1_P_Nr=21
      SK1_Fzg_Typ=0
      ;Zange schliessen
      $OUT[O_BM1_FRGZYL]=TRUE
      $OUT[O_BM1_ZYL_R]=FALSE
      $OUT[O_BM1_ZYL_V]=TRUE
      ;Leckagenausgleich
      $OUT[O_BM1_LE_AR]=FALSE
      $OUT[O_BM1_LE_AV]=TRUE
    ENDIF
;
    IF ($OUT[O_BM1_ZYL_V] AND $IN[I_BM1_KAH_S] AND $FLAG[F_m_BM1_Einz]) THEN
      $OUT[O_BM1_FRGZYL]=FALSE
      $OUT[O_BM1_ZYL_V]=FALSE
      $OUT[O_BM1_LE_AV]=FALSE
    ENDIF
    ;
    ;BM 1 schliessen in Hand  mit Zustellhub
    ;Schiebezylinder ist Vor
    IF ($OUT[O_BM1_zu] AND $FLAG[F_m_BM1_Einz] AND NOT $FLAG[F_m_BM1_Dopp]  AND NOT $FLAG[F_m_BM2_Einz] AND NOT $FLAG[F_m_BM2_Dopp]) THEN
      SK1_P_Nr=21
      SK1_Fzg_Typ=0
      ;Zange schliessen
      $OUT[O_BM1_FRGZYL]=TRUE
      $OUT[O_BM1_ZYL_V]=TRUE
      $OUT[O_BM1_ZYL_R]=FALSE
      ;Leckagenausgleich
      $OUT[O_BM1_LE_AR]=FALSE
      $OUT[O_BM1_LE_AV]=TRUE
    ENDIF
;
    IF ($OUT[O_BM1_ZYL_V] AND $IN[I_BM1_KAH_S] AND $FLAG[F_m_BM1_Einz]) THEN
      $OUT[O_BM1_FRGZYL]=FALSE
      $OUT[O_BM1_ZYL_V]=FALSE
      $OUT[O_BM1_LE_AV]=FALSE
    ENDIF
;
    ;BM 1 Zustellhub schliessen in Hand
    IF($OUT[O_BM1_VorZu] AND NOT $FLAG[F_m_BM1_Einz] AND NOT $FLAG[F_m_BM2_Einz] AND $FLAG[F_m_BM1_Dopp] AND NOT $FLAG[F_m_BM2_Dopp]) THEN
      SK1_P_Nr=21
      SK1_Fzg_Typ=0
      ;Zange schliessen
      $OUT[O_BM1_FRGZYL]=TRUE
      $OUT[O_BM1_ZYL_R]=TRUE
      $OUT[O_BM1_ZYL_V]=FALSE
      $OUT[O_BM1_ZH_R]=FALSE
      $OUT[O_BM1_ZH_V]=TRUE
    ENDIF
    ;
    IF ($OUT[O_BM1_ZYL_R] AND $IN[I_BM1_KZH_V] AND $FLAG[F_m_BM1_Dopp]) THEN
      $OUT[O_BM1_FRGZYL]=FALSE
      $OUT[O_BM1_ZYL_R]=FALSE
      $OUT[O_BM1_ZYL_V]=FALSE
      $OUT[O_BM1_ZH_R]=FALSE
      $OUT[O_BM1_ZH_V]=FALSE
    ENDIF
    ;
    ;BM1 Schiebezylinder Vor in Hand
    IF($OUT[O_BM1_SchVor] AND NOT $FLAG[F_m_BM1_Einz] AND NOT $FLAG[F_m_BM2_Einz] AND $FLAG[F_m_BM1_Dopp] AND NOT $FLAG[F_m_BM2_Dopp] AND NOT $IN[I_BM1_KSD_E] ) THEN
      SK1_P_Nr=21
      SK1_Fzg_Typ=0
      ;Schiebezylinder vor
      $OUT[O_BM1_FRGZYL]=TRUE
      $OUT[O_BM1_SZYL_R]=FALSE
      $OUT[O_BM1_SZYL_V]=TRUE
    ENDIF
;
    IF ($OUT[O_BM1_SZYL_V] AND $IN[I_BM1_SZYL_V] AND $FLAG[F_m_BM1_Dopp] ) THEN
      $OUT[O_BM1_FRGZYL]=FALSE
      $OUT[O_BM1_SZYL_V]=FALSE
    ENDIF
;
    ;Oeffnen der Stanze BM1
    ;Schiebezylinder  Rueck BM1
    ;BM1 Oeffnen in Hand ohne Zustellhub
    IF ($OUT[O_BM1_auf] AND $FLAG[F_m_BM1_Einz] AND NOT $FLAG[F_m_BM2_Einz] AND NOT $FLAG[F_m_BM1_Dopp]AND NOT $FLAG[F_m_BM2_Dopp]) THEN
      SK1_P_Nr=21
      SK1_Fzg_Typ=0
      ;Zange oeffnen
      $OUT[O_BM1_FRGZYL]=TRUE
      $OUT[O_BM1_ZYL_V]=FALSE
      $OUT[O_BM1_ZYL_R]=TRUE
      ;Leckagenausgleich
      $OUT[O_BM1_LE_AR]=FALSE
      $OUT[O_BM1_LE_AV]=TRUE
    ENDIF
;
    IF ($OUT[O_BM1_ZYL_R] AND $IN[I_BM1_BZZH_O] AND $FLAG[F_m_BM1_Einz]) THEN
      $OUT[O_BM1_FRGZYL]=FALSE
      $OUT[O_BM1_ZYL_R]=FALSE
      $OUT[O_BM1_ZYL_V]=FALSE
      $OUT[O_BM1_LE_AV]=FALSE
    ENDIF
;
    ;BM 1 Oeffnen in Hand Komplett mit Zustellhub
    IF ($OUT[O_BM1_Auf] AND NOT $FLAG[F_m_BM1_Einz] AND NOT $FLAG[F_m_BM2_Einz] AND NOT $FLAG[F_m_BM2_Dopp] AND $FLAG[F_m_BM1_Dopp] ) THEN
      SK1_P_Nr=21
      SK1_Fzg_Typ=0
      ;Zange oeffnen
      $OUT[O_BM1_FRGZYL]=TRUE
      $OUT[O_BM1_ZYL_V]=FALSE
      $OUT[O_BM1_ZYL_R]=TRUE
      $OUT[O_BM1_ZH_V]=FALSE
      $OUT[O_BM1_ZH_R]=TRUE
      ;Leckagenausgleich
      $OUT[O_BM1_LE_AR]=FALSE
      $OUT[O_BM1_LE_AV]=TRUE
    ENDIF

    IF ($OUT[O_BM1_ZH_R] AND $IN[I_BM1_BZZH_O] AND $FLAG[F_m_BM1_Dopp]) THEN
     $OUT[O_BM1_FRGZYL]=FALSE
     $OUT[O_BM1_ZYL_R]=FALSE
     $OUT[O_BM1_LE_AV]=FALSE
     $OUT[O_BM1_ZYL_V]=FALSE
     $OUT[O_BM1_ZH_R]=FALSE
    ENDIF
;
    ;BM1 oeffnen in Hand Zustellhub
    IF ($OUT[O_BM1_VorAuf] AND NOT $FLAG[F_m_BM1_Einz] AND NOT $FLAG[F_m_BM2_Einz] AND NOT $FLAG[F_m_BM2_Dopp] AND $FLAG[F_m_BM1_Dopp]) THEN
      SK1_P_Nr=21
      SK1_Fzg_Typ=0
      ;Zange oeffnen
      $OUT[O_BM1_FRGZYL]=TRUE
      $OUT[O_BM1_ZYL_V]=FALSE
      $OUT[O_BM1_ZYL_R]=TRUE
      $OUT[O_BM1_ZH_V]=TRUE
      $OUT[O_BM1_ZH_R]=FALSE
      ;Leckagenausgleich
      $OUT[O_BM1_LE_AR]=FALSE
      $OUT[O_BM1_LE_AV]=TRUE
    ENDIF
;
    IF ($OUT[O_BM1_ZYL_R] AND $IN[I_BM1_KZH_V] AND $FLAG[F_m_BM1_Dopp]) THEN
      $OUT[O_BM1_FRGZYL]=FALSE
      $OUT[O_BM1_ZYL_R]=FALSE
      $OUT[O_BM1_LE_AV]=FALSE
      $OUT[O_BM1_ZH_V]=FALSE
    ENDIF
;
    ;BM 1 schiebezylinder Rueck in Hand
    IF ($OUT[O_BM1_SchRue] AND NOT $FLAG[F_m_BM1_Einz] AND NOT $FLAG[F_m_BM2_Einz] AND $FLAG[F_m_BM1_Dopp] AND NOT $FLAG[F_m_BM2_Dopp] AND NOT $IN[I_BM1_KAH_S]) THEN
      SK1_P_Nr=21
      SK1_Fzg_Typ=0
      ;Schiebezylinder vor
      $OUT[O_BM1_FRGZYL]=TRUE
      $OUT[O_BM1_SZYL_V]=FALSE
      $OUT[O_BM1_SZYL_R]=TRUE
    ENDIF
;
    IF ($OUT[O_BM1_SZYL_R] AND $IN[I_BM1_SZYL_R]) THEN
      $OUT[O_BM1_FRGZYL]=FALSE
      $OUT[O_BM1_SZYL_R]=FALSE
    ENDIF
;
 ENDIF
End
;
;FOLD LOOP Mutterbuckeln VW-V3
GLOBAL DEF BM2_LOOP( )
  IF $FLAG[F_m_BM2_Einz] OR $FLAG[F_m_BM2_Dopp] THEN
    MIT_BM2=TRUE
  ELSE
    MIT_BM2=FALSE
  ENDIF
  ;Ausgabe Fehlermeldungen
  IF MIT_BM2 THEN
   ;
   ;Sammelstoerung
  $OUT[O_BM2_Sammel]=$OUT[O_R_Auto] AND $COULD_START_MOTION AND ($OUT[O_SK2_Sammel] OR $FLAG[F_SK2_Sammel]) AND $timer_flag[TimerNr_Ein]
  ENDIF
;
 IF ($OUT[O_R_Hand] AND NOT $OUT[O_R_Auto] AND $OUT[O_R_RK100] AND NOT $OUT[O_R_Proz_akt] AND NOT $FLAG[F_R_RobMove]) THEN

    ;BM2 schliessen in Hand ohne Zustellhub
    IF ($OUT[O_BM2_zu] AND NOT $FLAG[F_m_BM2_Einz] AND $FLAG[F_m_BM2_Einz] AND NOT $FLAG[F_m_BM1_Dopp] AND NOT $FLAG[F_m_BM2_Dopp]) THEN
      SK2_P_Nr=21
      SK2_Fzg_Typ=0
      ;Zange schliessen
      $OUT[O_BM2_FRGZYL]=TRUE
      $OUT[O_BM2_ZYL_R]=FALSE
      $OUT[O_BM2_ZYL_V]=TRUE
      ;Leckagenausgleich
      $OUT[O_BM2_LE_AR]=FALSE
      $OUT[O_BM2_LE_AV]=TRUE
    ENDIF

    IF ($OUT[O_BM2_ZYL_V] AND $IN[I_BM2_KAH_S] AND $FLAG[F_m_BM2_Einz]) THEN
      $OUT[O_BM2_FRGZYL]=FALSE
      $OUT[O_BM2_ZYL_V]=FALSE
      $OUT[O_BM2_LE_AV]=FALSE
      $OUT[O_BM2_LE_AR]=FALSE
    ENDIF

    ;BM 2 schliessen in Hand mit Zustellhub
    ;Schiebezylinder ist Vor
    IF ($OUT[O_BM2_zu] AND NOT $FLAG[F_m_BM1_Einz] AND NOT $FLAG[F_m_BM1_Dopp] AND NOT $FLAG[F_m_BM2_Einz] AND $FLAG[F_m_BM2_Dopp]) THEN
      SK2_P_Nr=21
      SK2_Fzg_Typ=0
      ;Zange schliessen
      $OUT[O_BM2_FRGZYL]=TRUE
      $OUT[O_BM2_ZYL_V]=TRUE
      $OUT[O_BM2_ZYL_R]=FALSE
      ;Leckagenausgleich
      $OUT[O_BM2_LE_AR]=FALSE
      $OUT[O_BM2_LE_AV]=TRUE
    ENDIF

    IF ($OUT[O_BM2_ZYL_V] AND $IN[I_BM2_KAH_S] AND $FLAG[F_m_BM2_Dopp]) THEN
      $OUT[O_BM2_FRGZYL]=FALSE
      $OUT[O_BM2_ZYL_V]=FALSE
      $OUT[O_BM2_LE_AV]=FALSE
      $OUT[O_BM2_LE_AR]=FALSE
    ENDIF

    ;Oeffnen der Stanze BM1
    ;Schiebezylinder  Rueck BM1
    ;BM 2 Schiebezylinder Vor in Hand
    IF ($OUT[O_BM2_SchVor] AND NOT $FLAG[F_m_BM1_Einz] AND NOT $FLAG[F_m_BM2_Einz] AND NOT $FLAG[F_m_BM1_Dopp] AND $FLAG[F_m_BM2_Dopp] AND NOT $IN[I_BM2_KSD_E]) THEN
      SK2_P_Nr=21
      SK2_Fzg_Typ=0
      ;Schiebezylinder vor
      $OUT[O_BM2_FRGZYL]=TRUE
      $OUT[O_BM2_SZYL_R]=FALSE
      $OUT[O_BM2_SZYL_V]=TRUE
    ENDIF

    IF ($OUT[O_BM2_SZYL_V] AND $IN[I_BM2_SZYL_V] AND $FLAG[F_m_BM2_Dopp]) THEN
      $OUT[O_BM2_FRGZYL]=FALSE
      $OUT[O_BM2_SZYL_V]=FALSE
    ENDIF

    ;BM2  Zustellhub schliessen in Hand
    IF($OUT[O_BM2_VorZu] AND NOT $FLAG[F_m_BM1_Einz] AND NOT $FLAG[F_m_BM2_Einz] AND NOT $FLAG[F_m_BM1_Dopp] AND $FLAG[F_m_BM2_Dopp]) THEN
      SK2_P_Nr=21
      SK2_Fzg_Typ=0
      ;Zange schliessen
      $OUT[O_BM2_FRGZYL]=TRUE
      $OUT[O_BM2_ZYL_R]=TRUE
      $OUT[O_BM2_ZYL_V]=FALSE
      $OUT[O_BM2_ZH_R]=FALSE
      $OUT[O_BM2_ZH_V]=TRUE
    ENDIF
    ;
    IF ($OUT[O_BM2_ZYL_R] AND $IN[I_BM2_KZH_V] AND $FLAG[F_m_BM2_Dopp]) THEN
      $OUT[O_BM2_FRGZYL]=FALSE
      $OUT[O_BM2_ZYL_R]=FALSE
      $OUT[O_BM2_ZYL_V]=FALSE
      $OUT[O_BM2_ZH_R]=FALSE
      $OUT[O_BM2_ZH_V]=FALSE
    ENDIF
    ;
    ;BM2 Oeffnen in Hand ohne Zustellhub
    IF ($OUT[O_BM2_auf] AND $FLAG[F_m_BM2_Einz] AND $FLAG[F_m_BM2_Einz] AND NOT $FLAG[F_m_BM1_Dopp]) THEN
      SK2_P_Nr=21
      SK2_Fzg_Typ=0
      ;Zange oeffnen
      $OUT[O_BM2_FRGZYL]=TRUE
      $OUT[O_BM2_ZYL_V]=FALSE
      $OUT[O_BM2_ZYL_R]=TRUE
      ;Leckagenausgleich
      $OUT[O_BM2_LE_AR]=FALSE
      $OUT[O_BM2_LE_AV]=TRUE
    ENDIF
;
    IF ($OUT[O_BM2_ZYL_R] AND $IN[I_BM2_BZZH_O] AND $FLAG[F_m_BM2_Einz]) THEN
      $OUT[O_BM2_FRGZYL]=FALSE
      $OUT[O_BM2_ZYL_R]=FALSE
      $OUT[O_BM2_LE_AV]=FALSE
    ENDIF
;
    ;BM 2 Oeffnen in Hand Komplett mit Zustellhub
    IF ($OUT[O_BM2_Auf] AND NOT $FLAG[F_m_BM1_Einz] AND NOT $FLAG[F_m_BM2_Einz] AND $FLAG[F_m_BM2_Dopp] AND NOT $FLAG[F_m_BM1_Dopp]) THEN
      SK2_P_Nr=21
      SK2_Fzg_Typ=0
      ;Zange oeffnen
      $OUT[O_BM2_FRGZYL]=TRUE
      $OUT[O_BM2_ZYL_V]=FALSE
      $OUT[O_BM2_ZYL_R]=TRUE
      $OUT[O_BM2_ZH_V]=FALSE
      $OUT[O_BM2_ZH_R]=TRUE
      ;Leckagenausgleich
      $OUT[O_BM2_LE_AR]=FALSE
      $OUT[O_BM2_LE_AV]=TRUE
    ENDIF
;
    IF ($OUT[O_BM2_ZH_R] AND $IN[I_BM2_BZZH_O] AND $FLAG[F_m_BM2_Dopp]) THEN
      $OUT[O_BM2_FRGZYL]=FALSE
      $OUT[O_BM2_ZYL_R]=FALSE
      $OUT[O_BM2_LE_AV]=FALSE
      $OUT[O_BM2_ZYL_V]=FALSE
      $OUT[O_BM2_ZH_R]=FALSE
    ENDIF
;
    ;BM2 oeffnen in Hand Zustellhub
    IF ($OUT[O_BM2_VorAuf] AND NOT $FLAG[F_m_BM1_Einz] AND NOT $FLAG[F_m_BM2_Einz] AND NOT $FLAG[F_m_BM1_Dopp] AND $FLAG[F_m_BM2_Dopp]) THEN
      SK2_P_Nr=21
      SK2_Fzg_Typ=0
      ;Zange oeffnen
      $OUT[O_BM2_FRGZYL]=TRUE
      $OUT[O_BM2_ZYL_V]=FALSE
      $OUT[O_BM2_ZYL_R]=TRUE
      $OUT[O_BM2_ZH_V]=TRUE
      $OUT[O_BM2_ZH_R]=FALSE
      ;Leckagenausgleich
      $OUT[O_BM2_LE_AR]=FALSE
      $OUT[O_BM2_LE_AV]=TRUE
    ENDIF
;
    IF ($OUT[O_BM1_ZYL_R] AND $IN[I_BM1_KZH_V] AND $FLAG[F_m_BM2_Dopp]) THEN
      $OUT[O_BM2_FRGZYL]=FALSE
      $OUT[O_BM2_ZYL_R]=FALSE
      $OUT[O_BM2_LE_AV]=FALSE
      $OUT[O_BM2_ZH_V]=FALSE
    ENDIF
;
    ;BM2 Schiebezylinder Rueck in Hand
    IF ($OUT[O_BM2_SchRue] AND NOT $FLAG[F_m_BM1_Einz] AND NOT $FLAG[F_m_BM2_Einz] AND NOT $FLAG[F_m_BM1_Dopp] AND $FLAG[F_m_BM2_Dopp] AND NOT $IN[I_BM2_KAH_S]) THEN
      SK2_P_Nr=21
      SK2_Fzg_Typ=0
      ;Schiebezylinder vor
      $OUT[O_BM2_FRGZYL]=TRUE
      $OUT[O_BM2_SZYL_V]=FALSE
      $OUT[O_BM2_SZYL_R]=TRUE
    ENDIF
;
    IF ($OUT[O_BM2_SZYL_R] AND $IN[I_BM2_SZYL_R]) THEN
      $OUT[O_BM2_FRGZYL]=FALSE
      $OUT[O_BM2_SZYL_R]=FALSE
    ENDIF
  ENDIF
;
END
;
;~~~~~~~~~VW-Teil-Ende~~~~~~~~
;
;-----------------------------------------------------------
;FOLD Lebensbit SZ
DEF L_Bit_SZ(SZNr :IN)
;Setzen / Rueksetzen Lebensbit Roboter
INT SZNr
BOOL LBitSZ, LBitFault
INT RobTimer
BOOL ErrLBit, bRet
ErrLBit = FALSE
LBitFault=FALSE
;Setzen - Rucksetzen  des Lebensbit an Zangensteuerung
$OUT[LBitToSZ[SZNr]] = NOT $IN[LBitFromSZ[SZNr]]
RobTimer = $ROB_TIMER
IF $IN[LBitFromSZ[SZNr]] <> LBitState[SZNr] THEN
  LBitTimeCnt[SZNr] = RobTimer
ENDIF
IF (RobTimer - LBitTimeCnt[SZNr]) > 5000 THEN
  ErrLBit = TRUE
  ErrSZNr = SZNr
  SZ_LBitFeh[SZNr]=TRUE
ENDIF
LBitState[SZNr] = $IN[LBitFromSZ[SZNr]]
IF ErrLBit THEN
  S_Zangen_Msg(4,#StateMsg, ErrSZNr)
ELSE
  IF n_SZS_Handle[4]>-1 THEN
    bRet=Clear_KrlMsg(n_SZS_Handle[4])
    n_SZS_Handle[4]=-1
    ErrSZNr = -1
  ENDIF
  SZ_LBitFeh[SZNr]=FALSE
ENDIF
;
END
;ENDFOLD
;
;-----------------------------------------------------------
;FOLD Lebensbit Kombisteuerungen
DEF L_Bit_Kombi(SZNr :IN)
;Setzen / Rueksetzen Lebensbit Roboter
INT SZNr
BOOL LBitSZ, LBitFault
INT RobTimer
BOOL ErrLBit, bRet
ErrLBit = FALSE
LBitFault=FALSE
;Setzen - Rucksetzen  des Lebensbit an Zangensteuerung
$OUT[LBitToKS[SZNr]] = NOT $IN[LBitFromKS[SZNr]]
RobTimer = $ROB_TIMER
IF $IN[LBitFromKS[SZNr]] <> LBitState[SZNr] THEN
  LBitTimeCnt[SZNr] = RobTimer
ENDIF
IF (RobTimer - LBitTimeCnt[SZNr]) > 5000 THEN
  ErrLBit = TRUE
  ErrSZNr = SZNr
  SZ_LBitFeh[SZNr]=TRUE
ENDIF
LBitState[SZNr] = $IN[LBitFromKS[SZNr]]
IF ErrLBit THEN
  S_Zangen_Msg(4,#StateMsg, ErrSZNr)
ELSE
  IF n_SZS_Handle[4]>-1 THEN
    bRet=Clear_KrlMsg(n_SZS_Handle[4])
    n_SZS_Handle[4]=-1
    ErrSZNr = -1
  ENDIF
  SZ_LBitFeh[SZNr]=FALSE
ENDIF
;
END
;ENDFOLD
;-----------------------------------------------------------
;FOLD SZ_Meldungen
DEF S_Zangen_Msg(msg_nr :IN, MsgTyp :IN, SZNr :IN )
INT msg_nr, SZNr, Answer
DECL SZS_MsgType MsgTyp
DECL KrlMsg_T USER_MSG
DECL KrlMsgPar_T Par[3]
DECL KrlMsgOpt_T Opt
;
USER_MSG = { Modul[] "SZ_S_Msg", Nr -1, Msg_txt[] " "}
Opt = { VL_Stop FALSE, Clear_P_Reset TRUE, Log_To_DB TRUE }
Par[1] = { Par_type #Value, Par_txt[] " " }
;
IF Varstate("SZNr")==#initialized then
  SWITCH SZNr
    CASE 1
      Par[1] = { Par_type #Value, Par_int 1 }
    CASE 2
      Par[1] = { Par_type #Value, Par_int 2 }
    CASE 3
      Par[1] = { Par_type #Value, Par_int 3 }
    CASE 4
      Par[1] = { Par_type #Value, Par_int 4 }
    CASE 5
      Par[1] = { Par_type #Value, Par_int 5 }
    CASE 6
      Par[1] = { Par_type #Value, Par_int 6 }
    DEFAULT
      Par[1] = { Par_type #Value, Par_txt[] " " }
  ENDSWITCH
ELSE
  Par[1] = { Par_type #Value, Par_txt[] " " }
ENDIF
;
IF ((n_SZS_Handle[msg_nr]<0) OR (MsgTyp==#NotifyMsg) OR (MsgTyp==#QuitMsg)) THEN
  USER_MSG.Nr = msg_nr
  SWITCH msg_nr
    CASE 1
	   USER_MSG.MSG_TXT[]="SZ1 Zange ist referenziert"
    CASE 2
	   USER_MSG.MSG_TXT[]="SZ2 Zange ist referenziert"
    CASE 3
	   USER_MSG.MSG_TXT[]="SZ3 Zange ist referenziert"
    CASE 4
	   USER_MSG.MSG_TXT[]="Zange%1 :keine Antwort auf Lebensbit"
    CASE 5
	   USER_MSG.MSG_TXT[]=" "
    CASE 6
	   USER_MSG.MSG_TXT[]=" "
    CASE 7
	   USER_MSG.MSG_TXT[]=" "
    CASE 20
      USER_MSG.MSG_TXT[]="Ausgleich fuer Zangenfunktion abgebrochen, neu anwaehlen"
    CASE 21
      USER_MSG.MSG_TXT[]="Programmanwahl fuer Zangenfunktion erforderlich"
    CASE 22
      USER_MSG.MSG_TXT[]="Init mit Start+ fuer Zangenfunktion erforderlich"
    CASE 23
      USER_MSG.MSG_TXT[]="Teachfunktion nicht erlaubt, wenn kein SingleStep"
    CASE 24
      USER_MSG.MSG_TXT[]="Erst SAK fahren, dann Zangenfunktion"
    CASE 31
      USER_MSG.MSG_TXT[]="SZ1 Zange teachen, Start+ erforderlich"
    CASE 32
      USER_MSG.MSG_TXT[]="SZ1 Zange oeffnen, Start+ erforderlich"
    CASE 33
      USER_MSG.MSG_TXT[]="SZ1 Zange schliessen, Start+ erforderlich"
    CASE 34
      USER_MSG.MSG_TXT[]="SZ1 Zangenfunktion nicht zulaessig"
    CASE 35
      USER_MSG.MSG_TXT[]="SZ1 Zangenfunktion bereits aktiv, SAW fuer Abbruch"
    CASE 41
      USER_MSG.MSG_TXT[]="SZ2 Zange teachen, Start+ erforderlich"
    CASE 42
      USER_MSG.MSG_TXT[]="SZ2 Zange oeffnen, Start+ erforderlich"
    CASE 43
      USER_MSG.MSG_TXT[]="SZ2 Zange schliessen, Start+ erforderlich"
    CASE 44
      USER_MSG.MSG_TXT[]="SZ2 Zangenfunktion nicht zulaessig"
    CASE 45
      USER_MSG.MSG_TXT[]="SZ2 Zangenfunktion bereits aktiv, SAW fuer Abbruch"
    CASE 51
      USER_MSG.MSG_TXT[]="SZ3 Zange teachen, Start+ erforderlich"
    CASE 52
      USER_MSG.MSG_TXT[]="SZ3 Zange oeffnen, Start+ erforderlich"
    CASE 53
      USER_MSG.MSG_TXT[]="SZ3 Zange schliessen, Start+ erforderlich"
    CASE 54
      USER_MSG.MSG_TXT[]="SZ2 Zangenfunktion nicht zulaessig"
    CASE 55
      USER_MSG.MSG_TXT[]="SZ3 Zangenfunktion bereits aktiv, SAW fuer Abbruch"
    DEFAULT
	   USER_MSG.MSG_TXT[]="unbekannte Meldung"
  ENDSWITCH
  SWITCH MsgTyp
    CASE #StateMsg
      n_SZS_Handle[msg_nr] = Set_KrlMsg (#State, USER_MSG, Par[], Opt) ;Ausgabe Statusmeldung
    CASE #QuitMsg
      n_SZS_Handle[msg_nr] = Set_KrlMsg (#Quit, USER_MSG, Par[], Opt) ;Ausgabe Quittierungsmeldung
    CASE #NotifyMsg
      n_SZS_Handle[msg_nr] = Set_KrlMsg (#Notify, USER_MSG, Par[], Opt) ;Ausgabe Hinweismeldung
    DEFAULT
      n_SZS_Handle[msg_nr] = Set_KrlMsg (#Quit, USER_MSG, Par[], Opt) ;Ausgabe Quittierungsmeldung
  ENDSWITCH
ENDIF
END
;
;ENDFOLD (NZ Meldungen)

--- vw_sz_usr_s.dat ---
&ACCESS  RV
&PARAM DISKPATH = VW_User/Applikation/S_Zange
&PARAM TPVW_VERSION = 8.3.0
&REL 203
DEFDAT  vw_sz_usr_s PUBLIC
;
;*-----------------------------------------------------*
;*Technologiepaket S_Zangen                            *
;*                                                     *
;*Konzernstandard                                      *
;*Bearbeiter: W. Lehmeier I/PG-C61                     *
;*                                                     *
;* Erstellt am:                                        *
;* 2015.02.19 LE                                       *
;*                                                     *
;*-----------------------------------------------------*
;
;FOLD USER_Version
STRUC _Tech_S_Zangen CHAR Name[20],INT Datum
DECL _Tech_S_Zangen Tech_S_Zangen
;ENDFOLD
;
;FOLD Ausgleich durch Roboter
GLOBAL INT Ausgl_an_KF=564
GLOBAL BOOL GunBal_Halt=FALSE
GLOBAL BOOL TeachPos=FALSE
; Funktionsuebergabe Zangenfuktion S_Int an R_Int
GLOBAL INT R1AusgleichFunktion=0
GLOBAL INT F_o_Ausgl=710
GLOBAL INT ov_merk=75
;ENDFOLD
;
;FOLD SZ_AH mit Roboterkompensation
GLOBAL INT F_SZ_AH_KOMP=290
;ENDFOLD
;
;FOLD SZ Kraftvorgabe in Hand
GLOBAL INT M_Kraft_Soll=20
;ENDFOLD
;
;FOLD Zangenoeffnung pruefen
GLOBAL INT Mit_Anf_Pos=713
GLOBAL INT F_SZ_Anf_Pos=741
;ENDFOLD
;
;FOLD Q-Tool
GLOBAL BOOL MIT_Q_Tool=FALSE
;
GLOBAL INT F_m_Q_Tool=272
;
GLOBAL INT Q_T_SZ1_VW=0
GLOBAL INT Q_T_SZ1_Fe=0
GLOBAL INT Q_T_SZ1_kD=0
GLOBAL INT Q_T_SZ2_VW=0
GLOBAL INT Q_T_SZ2_Fe=0
GLOBAL INT Q_T_SZ2_kD=0
GLOBAL INT Q_T_SZ3_VW=0
GLOBAL INT Q_T_SZ3_Fe=0
GLOBAL INT Q_T_SZ3_kD=0
;
GLOBAL INT F_QT_SZ1_VW=261
GLOBAL INT F_QT_SZ1_Fe=262
GLOBAL INT F_QT_SZ1_kD=263
GLOBAL INT F_QT_SZ2_VW=264
GLOBAL INT F_QT_SZ2_Fe=265
GLOBAL INT F_QT_SZ2_kD=266
GLOBAL INT F_QT_SZ3_VW=267
GLOBAL INT F_QT_SZ3_Fe=268
GLOBAL INT F_QT_SZ3_kD=269
;ENDFOLD
;
;FOLD SZ 1-3 EK-Verschleiss mit Vorzeichen
GLOBAL BOOL MIT_Val_N=FALSE
;ENDFOLD
;
;FOLD Konfiguration Ein-Ausgaenge SZ1
;Uebergabe Zangencode
SIGNAL EZ1_ZCode $OUT[761]  TO $OUT[763]
;Uebergabe Sollposition Stosspunkten
SIGNAL Stos_sollPos $OUT[737]  TO $OUT[751]
;Uebergabe Istposition Stosspunkten
SIGNAL Stos_istPos $IN[737]  TO $IN[751]
;Uebergabe Istposition
SIGNAL sig1_istpos $IN[737]  TO $IN[751]
;Uebergabe Ausgleichswert
SIGNAL SZ1_sollaus $OUT[729]  TO $OUT[736]
;SZ1-Drucksollwert Uebergabe
SIGNAL SZ1_Kraft_Soll $OUT[721]  TO $OUT[728]
SIGNAL SK1_Kraft_Soll $IN[793]  TO $IN[800]
;Programm-Nr an SZ 1
SIGNAL Prog_Nr_SZ1 $OUT[769]  TO $OUT[776]
SIGNAL Fzg_Typ_SZ1 $OUT[777]  TO $OUT[784]
;Programm-Nr an SK1
SIGNAL SK1_P_Nr $OUT[801]  TO $OUT[816]
SIGNAL SK1_Fzg_Typ $OUT[817]  TO $OUT[824]
;
GLOBAL BOOL B_SZ1_n_Ref=FALSE
;
GLOBAL INT F_SZ1_Anw_SF=78
GLOBAL INT F_SZ1_Anw_NF=79
GLOBAL INT F_SZ1_FRG_FR=92
GLOBAL INT F_SZ1_Sammel=118
GLOBAL INT F_SZ1_Schliess=120
GLOBAL INT F_SZ1_m_Komp=121
GLOBAL INT F_SZ1_Kapp1=122
GLOBAL INT F_SZ1_Kapp2=123
GLOBAL INT F_SZ1_Kapp3=124
GLOBAL INT F_SZ1_Kapp4=125
GLOBAL INT F_SZ1_KW_vor=131
GLOBAL INT F_SZ1_Pos_iO=742
GLOBAL INT F_SZ1_Oeff_iO=745
;
GLOBAL INT I_SZ1_oh_Kra=129
GLOBAL INT I_SZ1_bereit=705
GLOBAL INT I_SZ1_Re_aus=707
GLOBAL INT I_SZ1_EK_io=709
GLOBAL INT I_SZ1_TPos_g=711
GLOBAL INT I_SZ1_Auto=713
GLOBAL INT I_SZ1_ref=714
GLOBAL INT I_SZ1_aktiv=715
GLOBAL INT I_SZ1_IPos_g=716
GLOBAL INT I_SZ1_auf=717
GLOBAL INT I_SZ1_zu=718
GLOBAL INT I_SZ1_AR=719
GLOBAL INT I_SZ1_Vorz=752
GLOBAL INT I_SZ1_LBit=753
GLOBAL INT I_SZ1_GCodW1=766
GLOBAL INT I_SZ1_GCodW2=767
GLOBAL INT I_SZ1_GCodW4=768
GLOBAL INT I_SZ1_W_SZ=769
GLOBAL INT I_SZ1_W_Schm=770
GLOBAL INT I_SZ1_F_Kraf=771
GLOBAL INT I_SZ1_F_Prog=772
GLOBAL INT I_SZ1_F_Ziel=773
GLOBAL INT I_SZ1_F_Baut=774
GLOBAL INT I_SZ1_F_schw=775
GLOBAL INT I_SZ1_F_Frae=776
GLOBAL INT I_SZ1_F_Kapp=777
GLOBAL INT I_SZ1_F_Geom=778
GLOBAL INT I_SZ1_F_Schl=779
GLOBAL INT I_SZ1_F_Ausg=780
GLOBAL INT I_SZ1_F_Steu=781
GLOBAL INT I_SZ1_F_Traf=782
GLOBAL INT I_SZ1_F_Mot=783
GLOBAL INT I_SZ1_Sammel=784
;
GLOBAL INT O_SZ1_F_Schl=131
GLOBAL INT O_SZ1_W_SZ=132
GLOBAL INT O_SZ1_W_Schm=133
GLOBAL INT O_SZ1_F_Kraf=134
GLOBAL INT O_SZ1_F_Prog=135
GLOBAL INT O_SZ1_F_Ziel=136
GLOBAL INT O_SZ1_F_Baut=137
GLOBAL INT O_SZ1_F_schw=138
GLOBAL INT O_SZ1_F_Frae=139
GLOBAL INT O_SZ1_F_Geom=140
GLOBAL INT O_SZ1_F_Ausg=141
GLOBAL INT O_SZ1_F_Steu=142
GLOBAL INT O_SZ1_F_Temp=143
GLOBAL INT O_SZ1_Sammel=144
GLOBAL INT O_SZ1_Fe_Res=705
GLOBAL INT O_SZ1_E_Mode=706
GLOBAL INT O_SZ1_Re_aus=707
GLOBAL INT O_SZ1_oh_Kra=708
GLOBAL INT O_SZ1_Mit_EK=709
GLOBAL INT O_SZ1_S_TPos=710
GLOBAL INT O_SZ1_TPos_u=711
GLOBAL INT O_SZ1_R_Hand=712
GLOBAL INT O_SZ1_R_Auto=713
GLOBAL INT O_SZ1_ref=714
GLOBAL INT O_SZ1_FRG=715
GLOBAL INT O_SZ1_SPos_g=716
GLOBAL INT O_SZ1_auf=717
GLOBAL INT O_SZ1_zu=718
GLOBAL INT O_SZ1_t_auf=719
GLOBAL INT O_SZ1_t_zu=720
GLOBAL INT O_SZ1_H_Bit=736
GLOBAL INT O_SZ1_LBit=753
GLOBAL INT O_SZ1_m_RKom=754
GLOBAL INT O_SZ1_KW_io=755
GLOBAL INT O_SZ1_MvFrae=756
GLOBAL INT O_SZ1_MnFrae=757
GLOBAL INT O_SZ1_FToBT=760
GLOBAL INT O_SZ1_Teach=4001
GLOBAL INT O_SZ1_D_Auf=4002
GLOBAL INT O_SZ1_Du_Zu=4003
;ENDFOLD
;
;FOLD Konfiguration Ein-Ausgaenge SZ2
;Uebergabe Zangencode
SIGNAL EZ2_ZCode $OUT[921]  TO $OUT[923]
;Uebergabe Sollposition
SIGNAL sig2_sollpos $OUT[897]  TO $OUT[911]
;Uebergabe Istposition
SIGNAL sig2_istpos $IN[897]  TO $IN[911]
;Uebergabe Ausgleichswert
SIGNAL SZ2_sollaus $OUT[889]  TO $OUT[896]
;SZ2-Drucksollwert Uebergabe
SIGNAL SZ2_Kraft_Soll $OUT[881]  TO $OUT[888]
SIGNAL SK2_Kraft_Soll $IN[953]  TO $IN[960]
;Programm-Nr an SZ 2
SIGNAL Prog_Nr_SZ2 $OUT[929]  TO $OUT[936]
SIGNAL Fzg_Typ_SZ2 $OUT[937]  TO $OUT[944]
;Programm-Nr an SK1
SIGNAL SK2_P_Nr $OUT[961]  TO $OUT[976]
SIGNAL SK2_Fzg_Typ $OUT[977]  TO $OUT[984]
;
GLOBAL BOOL B_SZ2_n_Ref=FALSE
;
GLOBAL INT F_SZ2_Anw_SF=138
GLOBAL INT F_SZ2_Anw_NF=139
GLOBAL INT F_SZ2_FRG_FR=148
GLOBAL INT F_SZ2_Sammel=156
GLOBAL INT F_SZ2_Schliess=158
GLOBAL INT F_SZ2_m_Komp=159
GLOBAL INT F_SZ2_Kapp=160
GLOBAL INT F_SZ2_KW_vor=165
GLOBAL INT F_SZ2_Pos_iO=743
GLOBAL INT F_SZ2_Oeff_iO=746
;
GLOBAL INT I_SZ2_oh_Kra=161
GLOBAL INT I_SZ2_bereit=4081
GLOBAL INT I_SZ2_Re_aus=867
GLOBAL INT I_SZ2_EK_io=869
GLOBAL INT I_SZ2_TPos_g=871
GLOBAL INT I_SZ2_Auto=873
GLOBAL INT I_SZ2_ref=874
GLOBAL INT I_SZ2_aktiv=4082
GLOBAL INT I_SZ2_IPos_g=4081
GLOBAL INT I_SZ2_auf=877
GLOBAL INT I_SZ2_zu=878
GLOBAL INT I_SZ2_AR=879
GLOBAL INT I_SZ2_Vorz=912
GLOBAL INT I_SZ2_LBit=913
GLOBAL INT I_SZ2_GCodW1=926
GLOBAL INT I_SZ2_GCodW2=927
GLOBAL INT I_SZ2_GCodW4=928
GLOBAL INT I_SZ2_W_SZ=929
GLOBAL INT I_SZ2_W_Schm=930
GLOBAL INT I_SZ2_F_Kraf=931
GLOBAL INT I_SZ2_F_Prog=932
GLOBAL INT I_SZ2_F_Ziel=4082
GLOBAL INT I_SZ2_F_Baut=934
GLOBAL INT I_SZ2_F_schw=935
GLOBAL INT I_SZ2_F_Frae=936
GLOBAL INT I_SZ2_F_Kapp=937
GLOBAL INT I_SZ2_F_Geom=938
GLOBAL INT I_SZ2_F_Schl=939
GLOBAL INT I_SZ2_F_Ausg=940
GLOBAL INT I_SZ2_F_Steu=941
GLOBAL INT I_SZ2_F_Traf=942
GLOBAL INT I_SZ2_F_Mot=943
GLOBAL INT I_SZ2_Sammel=944
;
GLOBAL INT O_SZ2_F_Schl=163
GLOBAL INT O_SZ2_W_SZ=164
GLOBAL INT O_SZ2_W_Schm=165
GLOBAL INT O_SZ2_F_Kraf=166
GLOBAL INT O_SZ2_F_Prog=167
GLOBAL INT O_SZ2_F_Ziel=168
GLOBAL INT O_SZ2_F_Baut=169
GLOBAL INT O_SZ2_F_schw=170
GLOBAL INT O_SZ2_F_Frae=171
GLOBAL INT O_SZ2_F_Geom=172
GLOBAL INT O_SZ2_F_Ausg=173
GLOBAL INT O_SZ2_F_Steu=174
GLOBAL INT O_SZ2_F_Temp=175
GLOBAL INT O_SZ2_Sammel=176
GLOBAL INT O_SZ2_Fe_Res=865
GLOBAL INT O_SZ2_E_Mode=866
GLOBAL INT O_SZ2_Re_aus=867
GLOBAL INT O_SZ2_oh_Kra=868
GLOBAL INT O_SZ2_Mit_EK=869
GLOBAL INT O_SZ2_S_TPos=870
GLOBAL INT O_SZ2_TPos_u=871
GLOBAL INT O_SZ2_R_Hand=872
GLOBAL INT O_SZ2_R_Auto=873
GLOBAL INT O_SZ2_ref=874
GLOBAL INT O_SZ2_FRG=3658
GLOBAL INT O_SZ2_SPos_g=3658
GLOBAL INT O_SZ2_auf=877
GLOBAL INT O_SZ2_zu=878
GLOBAL INT O_SZ2_t_auf=879
GLOBAL INT O_SZ2_t_zu=880
GLOBAL INT O_SZ2_H_Bit=896
GLOBAL INT O_SZ2_LBit=913
GLOBAL INT O_SZ2_m_RKom=914
GLOBAL INT O_SZ2_KW_io=915
GLOBAL INT O_SZ2_MvFrae=916
GLOBAL INT O_SZ2_MnFrae=917
GLOBAL INT O_SZ2_FToBT=920
GLOBAL INT O_SZ2_Teach=4004
GLOBAL INT O_SZ2_D_Auf=4005
GLOBAL INT O_SZ2_Du_Zu=4006
;ENDFOLD
;
;FOLD Konfiguration Ein-Ausgaenge SZ3
;Uebergabe Zangencode
SIGNAL EZ3_ZCode $OUT[1081]  TO $OUT[1083]
;Uebergabe Sollposition
SIGNAL sig3_sollpos $OUT[1057]  TO $OUT[1071]
;Uebergabe Istposition
SIGNAL sig3_istpos $IN[1057]  TO $IN[1071]
;Uebergabe Ausgleichswert
SIGNAL SZ3_sollaus $OUT[1049]  TO $OUT[1056]
;Drucksollwert Uebergabe
SIGNAL SZ3_Kraft_Soll $OUT[1041]  TO $OUT[1048]
SIGNAL SK3_Kraft_Soll $IN[1113]  TO $IN[1120]
;Programm-Nr an SZ 3
SIGNAL Prog_Nr_SZ3 $OUT[1089]  TO $OUT[1096]
SIGNAL Fzg_Typ_SZ3 $OUT[1097]  TO $OUT[1104]
;Programm-Nr an SK1
SIGNAL SK3_P_Nr $OUT[1121]  TO $OUT[1136]
SIGNAL SK3_Fzg_Typ $OUT[1137]  TO $OUT[1144]
;
GLOBAL BOOL B_SZ3_n_Ref=FALSE
;
GLOBAL INT F_SZ3_Anw_SF=174
GLOBAL INT F_SZ3_Anw_NF=175
GLOBAL INT F_SZ3_FRG_FR=184
GLOBAL INT F_SZ3_Sammel=192
GLOBAL INT F_SZ3_Schliess=194
GLOBAL INT F_SZ3_m_Komp=195
GLOBAL INT F_SZ3_Kapp=196
GLOBAL INT F_SZ3_KW_vor=201
GLOBAL INT F_m_SZ2_TO_3=724
GLOBAL INT F_SZ3_Pos_iO=744
GLOBAL INT F_SZ3_Oeff_iO=747
;
GLOBAL INT I_SZ3_oh_Kra=193
GLOBAL INT I_SZ3_bereit=4081
GLOBAL INT I_SZ3_Re_aus=1027
GLOBAL INT I_SZ3_EK_io=1029
GLOBAL INT I_SZ3_TPos_g=1031
GLOBAL INT I_SZ3_Auto=1033
GLOBAL INT I_SZ3_ref=1034
GLOBAL INT I_SZ3_aktiv=4082
GLOBAL INT I_SZ3_IPos_g=4081
GLOBAL INT I_SZ3_auf=1037
GLOBAL INT I_SZ3_zu=1038
GLOBAL INT I_SZ3_AR=1039
GLOBAL INT I_SZ3_Vorz=1072
GLOBAL INT I_SZ3_LBit=1073
GLOBAL INT I_SZ3_GCodW1=1086
GLOBAL INT I_SZ3_GCodW2=1087
GLOBAL INT I_SZ3_GCodW4=1088
GLOBAL INT I_SZ3_W_SZ=1089
GLOBAL INT I_SZ3_W_Schm=1090
GLOBAL INT I_SZ3_F_Kraf=1091
GLOBAL INT I_SZ3_F_Prog=1092
GLOBAL INT I_SZ3_F_Ziel=4082
GLOBAL INT I_SZ3_F_Baut=1094
GLOBAL INT I_SZ3_F_schw=1095
GLOBAL INT I_SZ3_F_Frae=1096
GLOBAL INT I_SZ3_F_Kapp=1097
GLOBAL INT I_SZ3_F_Geom=1098
GLOBAL INT I_SZ3_F_Schl=1099
GLOBAL INT I_SZ3_F_Ausg=1100
GLOBAL INT I_SZ3_F_Steu=1101
GLOBAL INT I_SZ3_F_Traf=1102
GLOBAL INT I_SZ3_F_Mot=1103
GLOBAL INT I_SZ3_Sammel=1104
;
GLOBAL INT O_SZ3_F_Schl=195
GLOBAL INT O_SZ3_W_SZ=196
GLOBAL INT O_SZ3_W_Schm=197
GLOBAL INT O_SZ3_F_Kraf=198
GLOBAL INT O_SZ3_F_Prog=199
GLOBAL INT O_SZ3_F_Ziel=200
GLOBAL INT O_SZ3_F_Baut=201
GLOBAL INT O_SZ3_F_schw=202
GLOBAL INT O_SZ3_F_Frae=203
GLOBAL INT O_SZ3_F_Geom=204
GLOBAL INT O_SZ3_F_Ausg=205
GLOBAL INT O_SZ3_F_Steu=206
GLOBAL INT O_SZ3_F_Temp=207
GLOBAL INT O_SZ3_Sammel=208
GLOBAL INT O_SZ3_Fe_Res=1025
GLOBAL INT O_SZ3_E_Mode=1026
GLOBAL INT O_SZ3_Re_aus=1027
GLOBAL INT O_SZ3_oh_Kra=1028
GLOBAL INT O_SZ3_Mit_EK=1029
GLOBAL INT O_SZ3_S_TPos=1030
GLOBAL INT O_SZ3_TPos_u=1031
GLOBAL INT O_SZ3_R_Hand=1032
GLOBAL INT O_SZ3_R_Auto=1033
GLOBAL INT O_SZ3_ref=1034
GLOBAL INT O_SZ3_FRG=3658
GLOBAL INT O_SZ3_SPos_g=3658
GLOBAL INT O_SZ3_auf=1037
GLOBAL INT O_SZ3_zu=1038
GLOBAL INT O_SZ3_t_auf=1039
GLOBAL INT O_SZ3_t_zu=1040
GLOBAL INT O_SZ3_H_Bit=1048
GLOBAL INT O_SZ3_LBit=1073
GLOBAL INT O_SZ3_m_RKom=1074
GLOBAL INT O_SZ3_KW_io=1075
GLOBAL INT O_SZ3_MvFrae=1076
GLOBAL INT O_SZ3_MnFrae=1077
GLOBAL INT O_SZ3_FToBT=1080
GLOBAL INT O_SZ3_Teach=4007
GLOBAL INT O_SZ3_D_Auf=4008
GLOBAL INT O_SZ3_Du_Zu=4009
;ENDFOLD
;
;FOLD Lebensbit SZ
BOOL LBitState[3]
LBitState[1]=FALSE
LBitState[2]=FALSE
LBitState[3]=FALSE
BOOL SZ_LBitFeh[3]
SZ_LBitFeh[1]=FALSE
SZ_LBitFeh[2]=FALSE
SZ_LBitFeh[3]=FALSE
;
;Lebensbit an Zangensteuerung --- Ausgaenge ---
INT LBitToSZ[3]
LBitToSZ[1]=753
LBitToSZ[2]=913
LBitToSZ[3]=1073
;Lebensbit von Zangensteuerung --- Eingaenge ---
INT LBitFromSZ[3]
LBitFromSZ[1]=753
LBitFromSZ[2]=913
LBitFromSZ[3]=1073
;
INT LBitTimeCnt[3]
LBitTimeCnt[1]=48127
LBitTimeCnt[2]=48128
LBitTimeCnt[3]=48128
INT ErrSZNr=-1
;ENDFOLD
;
;FOLD Kombisteuerungen
GLOBAL BOOL Mit_Komb_ST=FALSE
GLOBAL BOOL Mit_Komb_ST1=FALSE
GLOBAL BOOL Mit_Komb_ST2=FALSE
GLOBAL BOOL Mit_Komb_ST3=FALSE
GLOBAL BOOL Temp_Komb_1=FALSE
GLOBAL BOOL Temp_Komb_2=FALSE
GLOBAL BOOL Temp_Komb_3=FALSE
;
GLOBAL INT F_m_Komb_ST1=830
GLOBAL INT F_m_Komb_ST2=831
GLOBAL INT F_m_Komb_ST3=832
;
;Kombisteuerung 1
;Zangencode an Kombi 1
SIGNAL Kb1_ZCode $OUT[765]  TO $OUT[767]
;Programm-Nr an Kombi 1
SIGNAL Prog_Nr_Kb1 $OUT[785]  TO $OUT[800]
;
GLOBAL INT I_Kb1_o_Schw=130
GLOBAL INT I_Kb1_Protok=132
GLOBAL INT I_Kb1_FrAnf=722
GLOBAL INT I_Kb1_V_Stdm=731
GLOBAL INT I_Kb1_M_Stdm=786
GLOBAL INT I_Kb1_W_Folg=789
GLOBAL INT I_Kb1_Ph_nio=790
GLOBAL INT I_Kb1_Primae=791
GLOBAL INT I_Kb1_F_Stro=792
GLOBAL INT I_Kb1_F_Span=793
GLOBAL INT I_Kb1_24V=794
GLOBAL INT I_Kb1_Invert=795
GLOBAL INT I_Kb1_Sammel=800
;
GLOBAL INT O_Kb1_W_SZ=131
GLOBAL INT O_Kb1_W_Schm=132
GLOBAL INT O_Kb1_FrAnf=133
GLOBAL INT O_Kb1_V_Stdm=134
GLOBAL INT O_Kb1_M_Stdm=135
GLOBAL INT O_Kb1_F_Kraf=136
GLOBAL INT O_Kb1_F_Prog=137
GLOBAL INT O_Kb1_F_Ziel=138
GLOBAL INT O_Kb1_F_Baut=139
GLOBAL INT O_Kb1_F_schw=140
GLOBAL INT O_Kb1_F_Frae=141
GLOBAL INT O_Kb1_F_KaVe=142
GLOBAL INT O_Kb1_F_Geom=143
GLOBAL INT O_Kb1_Schlep=144
GLOBAL INT O_Kb1_F_Ausg=145
GLOBAL INT O_Kb1_F_Steu=146
GLOBAL INT O_Kb1_FT_Tra=147
GLOBAL INT O_Kb1_FT_Mot=148
GLOBAL INT O_Kb1_WPS_io=149
GLOBAL INT O_Kb1_WP_nio=150
GLOBAL INT O_Kb1_W_Folg=151
GLOBAL INT O_Kb1_Ph_nio=152
GLOBAL INT O_Kb1_Primae=153
GLOBAL INT O_Kb1_F_Stro=154
GLOBAL INT O_Kb1_F_Span=155
GLOBAL INT O_Kb1_24V=156
GLOBAL INT O_Kb1_Invert=157
GLOBAL INT O_Kb1_Sammel=160
GLOBAL INT O_Kb1_Fe_Res=705
GLOBAL INT O_Kb1_zu_o_S=719
GLOBAL INT O_Kb1_t_auf=720
GLOBAL INT O_Kb1_t_zu=721
GLOBAL INT O_Kb1_MvFrae=724
GLOBAL INT O_Kb1_MnFrae=725
GLOBAL INT O_Kb1_KW_io=727
GLOBAL INT O_Kb1_Protok=728
GLOBAL INT O_Kb1_m_Stro=730
GLOBAL INT O_Kb1_FToBT=736
;
;Kombisteuerung 2
;Zangencode an Kombi 2
SIGNAL Kb2_ZCode $OUT[925]  TO $OUT[927]
;Programm-Nr an Kombi 2
SIGNAL Prog_Nr_Kb2 $OUT[945]  TO $OUT[960]
;
GLOBAL INT I_Kb2_o_Schw=162
GLOBAL INT I_Kb2_Protok=164
GLOBAL INT I_Kb2_FrAnf=882
GLOBAL INT I_Kb2_V_Stdm=891
GLOBAL INT I_Kb2_M_Stdm=946
GLOBAL INT I_Kb2_W_Folg=949
GLOBAL INT I_Kb2_Ph_nio=950
GLOBAL INT I_Kb2_Primae=951
GLOBAL INT I_Kb2_F_Stro=952
GLOBAL INT I_Kb2_F_Span=953
GLOBAL INT I_Kb2_24V=954
GLOBAL INT I_Kb2_Invert=955
GLOBAL INT I_Kb2_Sammel=960
;
GLOBAL INT O_Kb2_W_SZ=163
GLOBAL INT O_Kb2_W_Schm=164
GLOBAL INT O_Kb2_FrAnf=165
GLOBAL INT O_Kb2_V_Stdm=166
GLOBAL INT O_Kb2_M_Stdm=167
GLOBAL INT O_Kb2_F_Kraf=168
GLOBAL INT O_Kb2_F_Prog=169
GLOBAL INT O_Kb2_F_Ziel=170
GLOBAL INT O_Kb2_F_Baut=171
GLOBAL INT O_Kb2_F_schw=172
GLOBAL INT O_Kb2_F_Frae=173
GLOBAL INT O_Kb2_F_KaVe=174
GLOBAL INT O_Kb2_F_Geom=175
GLOBAL INT O_Kb2_Schlep=176
GLOBAL INT O_Kb2_F_Ausg=177
GLOBAL INT O_Kb2_F_Steu=178
GLOBAL INT O_Kb2_FT_Tra=179
GLOBAL INT O_Kb2_FT_Mot=180
GLOBAL INT O_Kb2_WPS_io=181
GLOBAL INT O_Kb2_WP_nio=182
GLOBAL INT O_Kb2_W_Folg=183
GLOBAL INT O_Kb2_Ph_nio=184
GLOBAL INT O_Kb2_Primae=185
GLOBAL INT O_Kb2_F_Stro=186
GLOBAL INT O_Kb2_F_Span=187
GLOBAL INT O_Kb2_24V=188
GLOBAL INT O_Kb2_Invert=189
GLOBAL INT O_Kb2_Sammel=192
GLOBAL INT O_Kb2_Fe_Res=865
GLOBAL INT O_Kb2_zu_o_S=879
GLOBAL INT O_Kb2_t_auf=880
GLOBAL INT O_Kb2_t_zu=881
GLOBAL INT O_Kb2_MvFrae=884
GLOBAL INT O_Kb2_MnFrae=885
GLOBAL INT O_Kb2_KW_io=887
GLOBAL INT O_Kb2_Protok=888
GLOBAL INT O_Kb2_m_Stro=890
GLOBAL INT O_Kb2_FToBT=896
;
;Kombisteuerung 3
;Zangencode an Kombi 3
SIGNAL Kb3_ZCode $OUT[1085]  TO $OUT[1087]
;Programm-Nr an Kombi 3
SIGNAL Prog_Nr_Kb3 $OUT[1105]  TO $OUT[1120]
;
GLOBAL INT I_Kb3_o_Schw=194
GLOBAL INT I_Kb3_Protok=196
GLOBAL INT I_Kb3_FrAnf=1042
GLOBAL INT I_Kb3_V_Stdm=1051
GLOBAL INT I_Kb3_M_Stdm=1106
GLOBAL INT I_Kb3_W_Folg=1109
GLOBAL INT I_Kb3_Ph_nio=1110
GLOBAL INT I_Kb3_Primae=1111
GLOBAL INT I_Kb3_F_Stro=1112
GLOBAL INT I_Kb3_F_Span=1113
GLOBAL INT I_Kb3_24V=1114
GLOBAL INT I_Kb3_Invert=1115
GLOBAL INT I_Kb3_Sammel=1120
;
GLOBAL INT O_Kb3_W_SZ=195
GLOBAL INT O_Kb3_W_Schm=196
GLOBAL INT O_Kb3_FrAnf=197
GLOBAL INT O_Kb3_V_Stdm=198
GLOBAL INT O_Kb3_M_Stdm=199
GLOBAL INT O_Kb3_F_Kraf=200
GLOBAL INT O_Kb3_F_Prog=201
GLOBAL INT O_Kb3_F_Ziel=202
GLOBAL INT O_Kb3_F_Baut=203
GLOBAL INT O_Kb3_F_schw=204
GLOBAL INT O_Kb3_F_Frae=205
GLOBAL INT O_Kb3_F_KaVe=206
GLOBAL INT O_Kb3_F_Geom=207
GLOBAL INT O_Kb3_Schlep=208
GLOBAL INT O_Kb3_F_Ausg=209
GLOBAL INT O_Kb3_F_Steu=210
GLOBAL INT O_Kb3_FT_Tra=211
GLOBAL INT O_Kb3_FT_Mot=212
GLOBAL INT O_Kb3_WPS_io=213
GLOBAL INT O_Kb3_WP_nio=214
GLOBAL INT O_Kb3_W_Folg=215
GLOBAL INT O_Kb3_Ph_nio=216
GLOBAL INT O_Kb3_Primae=217
GLOBAL INT O_Kb3_F_Stro=218
GLOBAL INT O_Kb3_F_Span=219
GLOBAL INT O_Kb3_24V=220
GLOBAL INT O_Kb3_Invert=221
GLOBAL INT O_Kb3_Sammel=224
GLOBAL INT O_Kb3_Fe_Res=1025
GLOBAL INT O_Kb3_zu_o_S=1039
GLOBAL INT O_Kb3_t_auf=1040
GLOBAL INT O_Kb3_t_zu=1041
GLOBAL INT O_Kb3_MvFrae=1044
GLOBAL INT O_Kb3_MnFrae=1045
GLOBAL INT O_Kb3_KW_io=1047
GLOBAL INT O_Kb3_Protok=1048
GLOBAL INT O_Kb3_m_Stro=1050
GLOBAL INT O_Kb3_FToBT=1056
;
;Lebensbit an Kombisteuerung --- Ausgaenge ---
INT LBitToKS[3]
LBitToKS[1]=729
LBitToKS[2]=889
LBitToKS[3]=1049
;Lebensbit von Kombisteuerung --- Eingaenge ---
INT LBitFromKS[3]
LBitFromKS[1]=729
LBitFromKS[2]=889
LBitFromKS[3]=1049
;ENDFOLD
;
;~~~~~~~~~VW-Teil-Anfang~~~~~~~~
;
;FOLD Mutternbuckeln 1 VW-Variante V3
GLOBAL BOOL MIT_BM1=FALSE
;
GLOBAL INT F_BM1_Sammel=208
GLOBAL INT F_m_BM1_Einz=211
GLOBAL INT F_m_BM1_Dopp=212
;
GLOBAL INT I_BM1_o_Proz=161
;
GLOBAL INT O_BM1_P_akt=161
GLOBAL INT O_BM1_nio=162
GLOBAL INT O_BM1_Mat=165
GLOBAL INT O_BM1_nBerei=167
GLOBAL INT O_BM1_Sammel=168
GLOBAL CONST INT O_BM1_FRGZYL=2705
GLOBAL CONST INT O_BM1_ZYL_R=2706
GLOBAL CONST INT O_BM1_ZYL_V=2707
GLOBAL CONST INT O_BM1_LE_AV=2708
GLOBAL CONST INT O_BM1_LE_AR=2709
GLOBAL CONST INT O_BM1_SZYL_R=2711
GLOBAL CONST INT O_BM1_SZYL_V=2712
GLOBAL CONST INT O_BM1_ZH_R=2719
GLOBAL CONST INT O_BM1_ZH_V=2720
GLOBAL CONST INT O_BM1_zu=4011
GLOBAL CONST INT O_BM1_Auf=4010
GLOBAL CONST INT O_BM1_VorAuf=4014
GLOBAL CONST INT O_BM1_VorZu=4015
GLOBAL CONST INT O_BM1_SchVor=4018
GLOBAL CONST INT O_BM1_SchRue=4019

GLOBAL CONST INT I_BM1_BZZH_O=2706
GLOBAL CONST INT I_BM1_KSD_E=2707
GLOBAL CONST INT I_BM1_KAH_S=2708
GLOBAL CONST INT I_BM1_KZH_V=2710
GLOBAL CONST INT I_BM1_SZYL_R=2711
GLOBAL CONST INT I_BM1_SZYL_V=2712

GLOBAL CONST INT F_R_RobMove=984
;ENDFOLD
;
;FOLD Mutternbuckeln 2 VW-Variante V3
GLOBAL BOOL MIT_BM2=FALSE
;
GLOBAL INT F_BM2_Sammel=218
GLOBAL INT F_m_BM2_Einz=222
GLOBAL INT F_m_BM2_Dopp=223
;
GLOBAL INT I_BM2_o_Proz=201
;
GLOBAL INT O_BM2_P_akt=201
GLOBAL INT O_BM2_nio=202
GLOBAL INT O_BM2_Mat=205
GLOBAL INT O_BM2_nBerei=207
GLOBAL INT O_BM2_Sammel=208
;
GLOBAL CONST INT O_BM2_FRGZYL=2721
GLOBAL CONST INT O_BM2_ZYL_R=2722
GLOBAL CONST INT O_BM2_ZYL_V=2723
GLOBAL CONST INT O_BM2_LE_AV=2724
GLOBAL CONST INT O_BM2_LE_AR=2725
GLOBAL CONST INT O_BM2_SZYL_R=2727
GLOBAL CONST INT O_BM2_SZYL_V=2728
GLOBAL CONST INT O_BM2_ZH_R=2735
GLOBAL CONST INT O_BM2_ZH_V=2736
GLOBAL CONST INT O_BM2_zu=4013
GLOBAL CONST INT O_BM2_Auf=4012
GLOBAL CONST INT O_BM2_VorAuf=4016
GLOBAL CONST INT O_BM2_VorZu=4017
GLOBAL CONST INT O_BM2_SchVor=4020
GLOBAL CONST INT O_BM2_SchRue=4021

GLOBAL CONST INT I_BM2_BZZH_O=2722
GLOBAL CONST INT I_BM2_KSD_E=2723
GLOBAL CONST INT I_BM2_KAH_S=2724
GLOBAL CONST INT I_BM2_KZH_V=2726
GLOBAL CONST INT I_BM2_SZYL_R=2727
GLOBAL CONST INT I_BM2_SZYL_V=2728
;
;ENDFOLD
;
;~~~~~~~~~VW-Teil-Ende~~~~~~~~
;
;FOLD Meldungsausgabe
ENUM SZS_MsgType StateMsg,QuitMsg,NotifyMsg
GLOBAL INT n_SZS_Handle[100]
GLOBAL INT n_SZR_Handle[100]
INT nMsgNum=0
INT RemMsgNum=0
;ENDFOLD
;
ENDDAT
